   DATA[823,17] := 1.0;
   DATA[823,18] := 1.0;
   DATA[823,19] := 1.0;
   DATA[823,20] := 148.808;
   DATA[823,21] := 155.5755;
   DATA[823,22] := 1.717489;
   DATA[823,23] := 970.0205;
   DATA[823,24] := 2.0;
   DATA[823,25] := 2.0;
   DATA[823,26] := 7.878942;
   DATA[823,27] := 144.7578;
   DATA[823,28] := 263.0415;
   DATA[823,29] := 12.11228;
   DATA[823,30] := 1.72507;
   DATA[823,31] := 1.291918;
   DATA[823,32] := 0.7352687;
   DATA[823,33] := 0.3083624;
   DATA[823,34] := 2.0;
   DATA[823,35] := 250.5608;
   DATA[823,36] := 1.730048;
   DATA[823,37] := 189.4386;
   DATA[823,38] := 0.000128152;
   DATA[823,39] := 1.0;
   DATA[824,0] := 2.535311;
   DATA[824,1] := 568.1444;
   DATA[824,2] := 2.0;
   DATA[824,3] := 1.0;
   DATA[824,4] := 262.3366;
   DATA[824,5] := 8.46533;
   DATA[824,6] := 315.1243;
   DATA[824,8] := 1.0;
   DATA[824,9] := 1.0;
   DATA[824,10] := 1.0;
   DATA[824,11] := 2.032781;
   DATA[824,13] := 1010.118;
   DATA[824,14] := 1.0;
   DATA[824,15] := 1.0;
   DATA[824,16] := 1.0;
   DATA[824,17] := 1.0;
   DATA[824,18] := 1.0;
   DATA[824,19] := 1.0;
   DATA[824,20] := 148.808;
   DATA[824,21] := 155.5755;
   DATA[824,22] := 1.717489;
   DATA[824,23] := 970.0974;
   DATA[824,24] := 2.0;
   DATA[824,25] := 2.0;
   DATA[824,26] := 7.878942;
   DATA[824,27] := 144.7578;
   DATA[824,28] := 263.0415;
   DATA[824,29] := 12.11228;
   DATA[824,30] := 1.72507;
   DATA[824,31] := 1.291533;
   DATA[824,32] := 0.7352687;
   DATA[824,33] := 0.3083624;
   DATA[824,34] := 2.0;
   DATA[824,35] := 250.5768;
   DATA[824,36] := 1.730048;
   DATA[824,37] := 189.4386;
   DATA[824,38] := 0.000128152;
   DATA[824,39] := 1.0;
   DATA[825,0] := 2.535311;
   DATA[825,1] := 569.5575;
   DATA[825,2] := 2.0;
   DATA[825,3] := 1.0;
   DATA[825,4] := 262.3366;
   DATA[825,5] := 8.46533;
   DATA[825,6] := 315.1243;
   DATA[825,8] := 1.0;
   DATA[825,9] := 1.0;
   DATA[825,10] := 1.0;
   DATA[825,11] := 2.032781;
   DATA[825,13] := 1010.158;
   DATA[825,14] := 1.0;
   DATA[825,15] := 1.0;
   DATA[825,16] := 1.0;
   DATA[825,17] := 1.0;
   DATA[825,18] := 1.0;
   DATA[825,19] := 1.0;
   DATA[825,20] := 148.808;
   DATA[825,21] := 155.5755;
   DATA[825,22] := 1.717489;
   DATA[825,23] := 969.3668;
   DATA[825,24] := 2.0;
   DATA[825,25] := 2.0;
   DATA[825,26] := 7.878942;
   DATA[825,27] := 144.7578;
   DATA[825,28] := 263.0415;
   DATA[825,29] := 11.92002;
   DATA[825,30] := 1.72507;
   DATA[825,31] := 1.274881;
   DATA[825,32] := 0.7352687;
   DATA[825,33] := 0.3071454;
   DATA[825,34] := 2.0;
   DATA[825,35] := 250.721;
   DATA[825,36] := 1.730048;
   DATA[825,37] := 189.4386;
   DATA[825,38] := 0.000128152;
   DATA[825,39] := 1.0;
   DATA[826,0] := 2.544278;
   DATA[826,1] := 570.3426;
   DATA[826,2] := 2.0;
   DATA[826,3] := 1.0;
   DATA[826,4] := 262.3366;
   DATA[826,5] := 8.46533;
   DATA[826,6] := 315.1243;
   DATA[826,8] := 1.0;
   DATA[826,9] := 1.0;
   DATA[826,10] := 1.0;
   DATA[826,11] := 2.032781;
   DATA[826,13] := 1010.478;
   DATA[826,14] := 1.0;
   DATA[826,15] := 1.0;
   DATA[826,16] := 1.0;
   DATA[826,17] := 1.0;
   DATA[826,18] := 1.0;
   DATA[826,19] := 1.0;
   DATA[826,20] := 148.808;
   DATA[826,21] := 155.5755;
   DATA[826,22] := 1.717489;
   DATA[826,23] := 969.2515;
   DATA[826,24] := 2.0;
   DATA[826,25] := 2.0;
   DATA[826,26] := 7.878942;
   DATA[826,27] := 144.7578;
   DATA[826,28] := 263.0415;
   DATA[826,29] := 11.92002;
   DATA[826,30] := 1.72789;
   DATA[826,31] := 1.27898;
   DATA[826,32] := 0.7352687;
   DATA[826,33] := 0.3069532;
   DATA[826,34] := 2.0;
   DATA[826,35] := 250.721;
   DATA[826,36] := 1.730048;
   DATA[826,37] := 189.4386;
   DATA[826,38] := 0.000128152;
   DATA[826,39] := 1.0;
   DATA[827,0] := 2.547161;
   DATA[827,1] := 570.9706;
   DATA[827,2] := 2.0;
   DATA[827,3] := 1.0;
   DATA[827,4] := 262.3366;
   DATA[827,5] := 8.46533;
   DATA[827,6] := 315.1243;
   DATA[827,8] := 1.0;
   DATA[827,9] := 1.0;
   DATA[827,10] := 1.0;
   DATA[827,11] := 2.032781;
   DATA[827,13] := 1010.358;
   DATA[827,14] := 1.0;
   DATA[827,15] := 1.0;
   DATA[827,16] := 1.0;
   DATA[827,17] := 1.0;
   DATA[827,18] := 1.0;
   DATA[827,19] := 1.0;
   DATA[827,20] := 148.808;
   DATA[827,21] := 155.5755;
   DATA[827,22] := 1.719156;
   DATA[827,23] := 969.0208;
   DATA[827,24] := 2.0;
   DATA[827,25] := 2.0;
   DATA[827,26] := 7.878942;
   DATA[827,27] := 144.7578;
   DATA[827,28] := 263.0415;
   DATA[827,29] := 11.92002;
   DATA[827,30] := 1.728147;
   DATA[827,31] := 1.282183;
   DATA[827,32] := 0.7352687;
   DATA[827,33] := 0.3069532;
   DATA[827,34] := 2.0;
   DATA[827,35] := 250.721;
   DATA[827,36] := 1.730048;
   DATA[827,37] := 189.4386;
   DATA[827,38] := 0.000128152;
   DATA[827,39] := 1.0;
   DATA[828,0] := 2.547161;
   DATA[828,1] := 572.2659;
   DATA[828,2] := 2.0;
   DATA[828,3] := 1.0;
   DATA[828,4] := 262.3366;
   DATA[828,5] := 8.46533;
   DATA[828,6] := 315.1243;
   DATA[828,8] := 1.0;
   DATA[828,9] := 1.0;
   DATA[828,10] := 1.0;
   DATA[828,11] := 2.032781;
   DATA[828,13] := 1010.879;
   DATA[828,14] := 1.0;
   DATA[828,15] := 1.0;
   DATA[828,16] := 1.0;
   DATA[828,17] := 1.0;
   DATA[828,18] := 1.0;
   DATA[828,19] := 1.0;
   DATA[828,20] := 148.808;
   DATA[828,21] := 155.5755;
   DATA[828,22] := 1.719156;
   DATA[828,23] := 968.3671;
   DATA[828,24] := 2.0;
   DATA[828,25] := 2.0;
   DATA[828,26] := 7.878942;
   DATA[828,27] := 144.7578;
   DATA[828,28] := 263.0415;
   DATA[828,29] := 11.92002;
   DATA[828,30] := 1.728147;
   DATA[828,31] := 1.282183;
   DATA[828,32] := 0.7352687;
   DATA[828,33] := 0.3069532;
   DATA[828,34] := 2.0;
   DATA[828,35] := 250.721;
   DATA[828,36] := 1.730048;
   DATA[828,37] := 189.4386;
   DATA[828,38] := 0.000128152;
   DATA[828,39] := 1.0;
   DATA[829,0] := 2.547161;
   DATA[829,1] := 572.7762;
   DATA[829,2] := 2.0;
   DATA[829,3] := 1.0;
   DATA[829,4] := 262.3366;
   DATA[829,5] := 8.46533;
   DATA[829,6] := 315.1243;
   DATA[829,8] := 1.0;
   DATA[829,9] := 1.0;
   DATA[829,10] := 1.0;
   DATA[829,11] := 2.032781;
   DATA[829,13] := 1010.558;
   DATA[829,14] := 1.0;
   DATA[829,15] := 1.0;
   DATA[829,16] := 1.0;
   DATA[829,17] := 1.0;
   DATA[829,18] := 1.0;
   DATA[829,19] := 1.0;
   DATA[829,20] := 148.808;
   DATA[829,21] := 155.8062;
   DATA[829,22] := 1.719156;
   DATA[829,23] := 967.9056;
   DATA[829,24] := 2.0;
   DATA[829,25] := 2.0;
   DATA[829,26] := 7.878942;
   DATA[829,27] := 144.7578;
   DATA[829,28] := 263.0415;
   DATA[829,29] := 11.92002;
   DATA[829,30] := 1.729557;
   DATA[829,31] := 1.282183;
   DATA[829,32] := 0.7352687;
   DATA[829,33] := 0.3065689;
   DATA[829,34] := 2.0;
   DATA[829,35] := 250.721;
   DATA[829,36] := 1.730048;
   DATA[829,37] := 189.4386;
   DATA[829,38] := 0.000128152;
   DATA[829,39] := 1.0;
   DATA[830,0] := 2.547161;
   DATA[830,1] := 573.2473;
   DATA[830,2] := 2.0;
   DATA[830,3] := 1.0;
   DATA[830,4] := 262.3366;
   DATA[830,5] := 8.46533;
   DATA[830,6] := 315.1243;
   DATA[830,8] := 1.0;
   DATA[830,9] := 1.0;
   DATA[830,10] := 1.0;
   DATA[830,11] := 2.032781;
   DATA[830,13] := 1010.919;
   DATA[830,14] := 1.0;
   DATA[830,15] := 1.0;
   DATA[830,16] := 1.0;
   DATA[830,17] := 1.0;
   DATA[830,18] := 1.0;
   DATA[830,19] := 1.0;
   DATA[830,20] := 148.808;
   DATA[830,21] := 155.8062;
   DATA[830,22] := 1.717746;
   DATA[830,23] := 967.4827;
   DATA[830,24] := 2.0;
   DATA[830,25] := 2.0;
   DATA[830,26] := 7.878942;
   DATA[830,27] := 144.7578;
   DATA[830,28] := 263.0415;
   DATA[830,29] := 11.92002;
   DATA[830,30] := 1.729557;
   DATA[830,31] := 1.282183;
   DATA[830,32] := 0.7352687;
   DATA[830,33] := 0.3079781;
   DATA[830,34] := 2.0;
   DATA[830,35] := 250.4967;
   DATA[830,36] := 1.730048;
   DATA[830,37] := 189.4386;
   DATA[830,38] := 0.000128152;
   DATA[830,39] := 1.0;
   DATA[831,0] := 2.547161;
   DATA[831,1] := 573.3258;
   DATA[831,2] := 2.0;
   DATA[831,3] := 1.0;
   DATA[831,4] := 262.3366;
   DATA[831,5] := 8.46533;
   DATA[831,6] := 315.1243;
   DATA[831,8] := 1.0;
   DATA[831,9] := 1.0;
   DATA[831,10] := 1.0;
   DATA[831,11] := 2.032781;
   DATA[831,13] := 1010.718;
   DATA[831,14] := 1.0;
   DATA[831,15] := 1.0;
   DATA[831,16] := 1.0;
   DATA[831,17] := 1.0;
   DATA[831,18] := 1.0;
   DATA[831,19] := 1.0;
   DATA[831,20] := 148.808;
   DATA[831,21] := 155.8062;
   DATA[831,22] := 1.717746;
   DATA[831,23] := 967.3289;
   DATA[831,24] := 2.0;
   DATA[831,25] := 2.0;
   DATA[831,26] := 7.878942;
   DATA[831,27] := 144.7578;
   DATA[831,28] := 263.0415;
   DATA[831,29] := 11.92002;
   DATA[831,30] := 1.729557;
   DATA[831,31] := 1.271935;
   DATA[831,32] := 0.7352687;
   DATA[831,33] := 0.3083624;
   DATA[831,34] := 2.0;
   DATA[831,35] := 250.4967;
   DATA[831,36] := 1.730048;
   DATA[831,37] := 189.4386;
   DATA[831,38] := 0.000128152;
   DATA[831,39] := 1.0;
   DATA[832,0] := 2.547161;
   DATA[832,1] := 574.4249;
   DATA[832,2] := 2.0;
   DATA[832,3] := 1.0;
   DATA[832,4] := 262.3366;
   DATA[832,5] := 8.46533;
   DATA[832,6] := 315.1243;
   DATA[832,8] := 1.0;
   DATA[832,9] := 1.0;
   DATA[832,10] := 1.0;
   DATA[832,11] := 2.032781;
   DATA[832,13] := 1011.039;
   DATA[832,14] := 1.0;
   DATA[832,15] := 1.0;
   DATA[832,16] := 1.0;
   DATA[832,17] := 1.0;
   DATA[832,18] := 1.0;
   DATA[832,19] := 1.0;
   DATA[832,20] := 148.808;
   DATA[832,21] := 155.5755;
   DATA[832,22] := 1.717746;
   DATA[832,23] := 966.9059;
   DATA[832,24] := 2.0;
   DATA[832,25] := 2.0;
   DATA[832,26] := 7.878942;
   DATA[832,27] := 144.7578;
   DATA[832,28] := 263.0415;
   DATA[832,29] := 11.92002;
   DATA[832,30] := 1.729557;
   DATA[832,31] := 1.279621;
   DATA[832,32] := 0.7352687;
   DATA[832,33] := 0.3083624;
   DATA[832,34] := 2.0;
   DATA[832,35] := 250.4967;
   DATA[832,36] := 1.730048;
   DATA[832,37] := 189.4386;
   DATA[832,38] := 0.000128152;
   DATA[832,39] := 1.0;
   DATA[833,0] := 2.555168;
   DATA[833,1] := 575.4454;
   DATA[833,2] := 2.0;
   DATA[833,3] := 1.0;
   DATA[833,4] := 262.3366;
   DATA[833,5] := 8.46533;
   DATA[833,6] := 315.1243;
   DATA[833,8] := 1.0;
   DATA[833,9] := 1.0;
   DATA[833,10] := 1.0;
   DATA[833,11] := 2.032781;
   DATA[833,13] := 1010.959;
   DATA[833,14] := 1.0;
   DATA[833,15] := 1.0;
   DATA[833,16] := 1.0;
   DATA[833,17] := 1.0;
   DATA[833,18] := 1.0;
   DATA[833,19] := 1.0;
   DATA[833,20] := 148.808;
   DATA[833,21] := 155.5755;
   DATA[833,22] := 1.717746;
   DATA[833,23] := 966.6752;
   DATA[833,24] := 2.0;
   DATA[833,25] := 2.0;
   DATA[833,26] := 7.878942;
   DATA[833,27] := 144.7578;
   DATA[833,28] := 263.0415;
   DATA[833,29] := 12.15073;
   DATA[833,30] := 1.729557;
   DATA[833,31] := 1.290893;
   DATA[833,32] := 0.7352687;
   DATA[833,33] := 0.3083624;
   DATA[833,34] := 2.0;
   DATA[833,35] := 250.737;
   DATA[833,36] := 1.730048;
   DATA[833,37] := 189.4386;
   DATA[833,38] := 0.000128152;
   DATA[833,39] := 1.0;
   DATA[834,0] := 2.555168;
   DATA[834,1] := 576.2697;
   DATA[834,2] := 2.0;
   DATA[834,3] := 1.0;
   DATA[834,4] := 262.3366;
   DATA[834,5] := 8.46533;
   DATA[834,6] := 315.1243;
   DATA[834,8] := 1.0;
   DATA[834,9] := 1.0;
   DATA[834,10] := 1.0;
   DATA[834,11] := 2.032781;
   DATA[834,13] := 1011.279;
   DATA[834,14] := 1.0;
   DATA[834,15] := 1.0;
   DATA[834,16] := 1.0;
   DATA[834,17] := 1.0;
   DATA[834,18] := 1.0;
   DATA[834,19] := 1.0;
   DATA[834,20] := 148.808;
   DATA[834,21] := 155.5755;
   DATA[834,22] := 1.717746;
   DATA[834,23] := 966.3676;
   DATA[834,24] := 2.0;
   DATA[834,25] := 2.0;
   DATA[834,26] := 7.878942;
   DATA[834,27] := 144.7578;
   DATA[834,28] := 263.0415;
   DATA[834,29] := 12.15073;
   DATA[834,30] := 1.729557;
   DATA[834,31] := 1.286153;
   DATA[834,32] := 0.7352687;
   DATA[834,33] := 0.3083624;
   DATA[834,34] := 2.0;
   DATA[834,35] := 250.737;
   DATA[834,36] := 1.730048;
   DATA[834,37] := 189.4386;
   DATA[834,38] := 0.000128152;
   DATA[834,39] := 1.0;
   DATA[835,0] := 2.555168;
   DATA[835,1] := 577.251;
   DATA[835,2] := 2.0;
   DATA[835,3] := 1.0;
   DATA[835,4] := 262.3366;
   DATA[835,5] := 8.46533;
   DATA[835,6] := 315.1243;
   DATA[835,8] := 1.0;
   DATA[835,9] := 1.0;
   DATA[835,10] := 1.0;
   DATA[835,11] := 2.032781;
   DATA[835,13] := 1011.079;
   DATA[835,14] := 1.0;
   DATA[835,15] := 1.0;
   DATA[835,16] := 1.0;
   DATA[835,17] := 1.0;
   DATA[835,18] := 1.0;
   DATA[835,19] := 1.0;
   DATA[835,20] := 148.808;
   DATA[835,21] := 155.5755;
   DATA[835,22] := 1.717746;
   DATA[835,23] := 965.7139;
   DATA[835,24] := 2.0;
   DATA[835,25] := 2.0;
   DATA[835,26] := 7.878942;
   DATA[835,27] := 144.7578;
   DATA[835,28] := 263.0415;
   DATA[835,29] := 12.15073;
   DATA[835,30] := 1.7293;
   DATA[835,31] := 1.288715;
   DATA[835,32] := 0.7352687;
   DATA[835,33] := 0.3083624;
   DATA[835,34] := 2.0;
   DATA[835,35] := 250.737;
   DATA[835,36] := 1.730048;
   DATA[835,37] := 189.6949;
   DATA[835,38] := 0.000128152;
   DATA[835,39] := 1.0;
   DATA[836,0] := 2.555168;
   DATA[836,1] := 577.8006;
   DATA[836,2] := 2.0;
   DATA[836,3] := 1.0;
   DATA[836,4] := 262.3366;
   DATA[836,5] := 8.46533;
   DATA[836,6] := 315.1243;
   DATA[836,8] := 1.0;
   DATA[836,9] := 1.0;
   DATA[836,10] := 1.0;
   DATA[836,11] := 2.032781;
   DATA[836,13] := 1011.079;
   DATA[836,14] := 1.0;
   DATA[836,15] := 1.0;
   DATA[836,16] := 1.0;
   DATA[836,17] := 1.0;
   DATA[836,18] := 1.0;
   DATA[836,19] := 1.0;
   DATA[836,20] := 148.808;
   DATA[836,21] := 155.5755;
   DATA[836,22] := 1.718515;
   DATA[836,23] := 965.3294;
   DATA[836,24] := 2.0;
   DATA[836,25] := 2.0;
   DATA[836,26] := 7.878942;
   DATA[836,27] := 144.7578;
   DATA[836,28] := 263.0415;
   DATA[836,29] := 12.15073;
   DATA[836,30] := 1.7293;
   DATA[836,31] := 1.281542;
   DATA[836,32] := 0.7352687;
   DATA[836,33] := 0.3083624;
   DATA[836,34] := 2.0;
   DATA[836,35] := 250.8972;
   DATA[836,36] := 1.730048;
   DATA[836,37] := 189.6949;
   DATA[836,38] := 0.000128152;
   DATA[836,39] := 1.0;
   DATA[837,0] := 2.555168;
   DATA[837,1] := 578.8212;
   DATA[837,2] := 2.0;
   DATA[837,3] := 1.0;
   DATA[837,4] := 262.3366;
   DATA[837,5] := 8.46533;
   DATA[837,6] := 315.1243;
   DATA[837,8] := 1.0;
   DATA[837,9] := 1.0;
   DATA[837,10] := 1.0;
   DATA[837,11] := 2.032781;
   DATA[837,13] := 1011.239;
   DATA[837,14] := 1.0;
   DATA[837,15] := 1.0;
   DATA[837,16] := 1.0;
   DATA[837,17] := 1.0;
   DATA[837,18] := 1.0;
   DATA[837,19] := 1.0;
   DATA[837,20] := 148.808;
   DATA[837,21] := 155.5755;
   DATA[837,22] := 1.720565;
   DATA[837,23] := 964.6373;
   DATA[837,24] := 2.0;
   DATA[837,25] := 2.0;
   DATA[837,26] := 7.878942;
   DATA[837,27] := 144.7578;
   DATA[837,28] := 263.0415;
   DATA[837,29] := 12.15073;
   DATA[837,30] := 1.7293;
   DATA[837,31] := 1.272192;
   DATA[837,32] := 0.7352687;
   DATA[837,33] := 0.3083624;
   DATA[837,34] := 2.0;
   DATA[837,35] := 250.8972;
   DATA[837,36] := 1.730048;
   DATA[837,37] := 189.6949;
   DATA[837,38] := 0.000128152;
   DATA[837,39] := 1.0;
   DATA[838,0] := 2.553886;
   DATA[838,1] := 579.724;
   DATA[838,2] := 2.0;
   DATA[838,3] := 1.0;
   DATA[838,4] := 262.3366;
   DATA[838,5] := 8.46533;
   DATA[838,6] := 315.1243;
   DATA[838,8] := 1.0;
   DATA[838,9] := 1.0;
   DATA[838,10] := 1.0;
   DATA[838,11] := 2.032781;
   DATA[838,13] := 1011.279;
   DATA[838,14] := 1.0;
   DATA[838,15] := 1.0;
   DATA[838,16] := 1.0;
   DATA[838,17] := 1.0;
   DATA[838,18] := 1.0;
   DATA[838,19] := 1.0;
   DATA[838,20] := 148.808;
   DATA[838,21] := 155.5755;
   DATA[838,22] := 1.720565;
   DATA[838,23] := 964.5988;
   DATA[838,24] := 2.0;
   DATA[838,25] := 2.0;
   DATA[838,26] := 7.878942;
   DATA[838,27] := 144.7578;
   DATA[838,28] := 263.0415;
   DATA[838,29] := 12.15073;
   DATA[838,30] := 1.7293;
   DATA[838,31] := 1.271679;
   DATA[838,32] := 0.736421;
   DATA[838,33] := 0.3083624;
   DATA[838,34] := 2.0;
   DATA[838,35] := 250.8972;
   DATA[838,36] := 1.730048;
   DATA[838,37] := 189.6949;
   DATA[838,38] := 0.000128152;
   DATA[838,39] := 1.0;
   DATA[839,0] := 2.54684;
   DATA[839,1] := 580.7053;
   DATA[839,2] := 2.0;
   DATA[839,3] := 1.0;
   DATA[839,4] := 262.3366;
   DATA[839,5] := 8.46533;
   DATA[839,6] := 315.1243;
   DATA[839,8] := 1.0;
   DATA[839,9] := 1.0;
   DATA[839,10] := 1.0;
   DATA[839,11] := 2.032781;
   DATA[839,13] := 1011.079;
   DATA[839,14] := 1.0;
   DATA[839,15] := 1.0;
   DATA[839,16] := 1.0;
   DATA[839,17] := 1.0;
   DATA[839,18] := 1.0;
   DATA[839,19] := 1.0;
   DATA[839,20] := 148.808;
   DATA[839,21] := 155.5755;
   DATA[839,22] := 1.720565;
   DATA[839,23] := 964.1758;
   DATA[839,24] := 2.0;
   DATA[839,25] := 2.0;
   DATA[839,26] := 7.878942;
   DATA[839,27] := 144.7578;
   DATA[839,28] := 263.0415;
   DATA[839,29] := 12.15073;
   DATA[839,30] := 1.7293;
   DATA[839,31] := 1.271551;
   DATA[839,32] := 0.7366771;
   DATA[839,33] := 0.3068891;
   DATA[839,34] := 2.0;
   DATA[839,35] := 250.8972;
   DATA[839,36] := 1.730048;
   DATA[839,37] := 189.5668;
   DATA[839,38] := 0.000128152;
   DATA[839,39] := 1.0;
   DATA[840,0] := 2.542356;
   DATA[840,1] := 581.2941;
   DATA[840,2] := 2.0;
   DATA[840,3] := 1.0;
   DATA[840,4] := 262.3366;
   DATA[840,5] := 8.46533;
   DATA[840,6] := 315.1243;
   DATA[840,8] := 1.0;
   DATA[840,9] := 1.0;
   DATA[840,10] := 1.0;
   DATA[840,11] := 2.026378;
   DATA[840,13] := 1010.879;
   DATA[840,14] := 1.0;
   DATA[840,15] := 1.0;
   DATA[840,16] := 1.0;
   DATA[840,17] := 1.0;
   DATA[840,18] := 1.0;
   DATA[840,19] := 1.0;
   DATA[840,20] := 148.808;
   DATA[840,21] := 155.5755;
   DATA[840,22] := 1.718771;
   DATA[840,23] := 963.7529;
   DATA[840,24] := 2.0;
   DATA[840,25] := 2.0;
   DATA[840,26] := 7.878942;
   DATA[840,27] := 144.7578;
   DATA[840,28] := 263.0415;
   DATA[840,29] := 12.15073;
   DATA[840,30] := 1.728019;
   DATA[840,31] := 1.271551;
   DATA[840,32] := 0.7373172;
   DATA[840,33] := 0.3068891;
   DATA[840,34] := 2.0;
   DATA[840,35] := 250.785;
   DATA[840,36] := 1.730048;
   DATA[840,37] := 189.4546;
   DATA[840,38] := 0.000128152;
   DATA[840,39] := 1.0;
   DATA[841,0] := 2.538833;
   DATA[841,1] := 581.5688;
   DATA[841,2] := 2.0;
   DATA[841,3] := 1.0;
   DATA[841,4] := 262.3366;
   DATA[841,5] := 8.46501;
   DATA[841,6] := 315.1243;
   DATA[841,8] := 1.0;
   DATA[841,9] := 1.0;
   DATA[841,10] := 1.0;
   DATA[841,11] := 2.026378;
   DATA[841,13] := 1011.159;
   DATA[841,14] := 1.0;
   DATA[841,15] := 1.0;
   DATA[841,16] := 1.0;
   DATA[841,17] := 1.0;
   DATA[841,18] := 1.0;
   DATA[841,19] := 1.0;
   DATA[841,20] := 148.808;
   DATA[841,21] := 155.5755;
   DATA[841,22] := 1.718771;
   DATA[841,23] := 963.4068;
   DATA[841,24] := 2.0;
   DATA[841,25] := 2.0;
   DATA[841,26] := 7.878942;
   DATA[841,27] := 144.7578;
   DATA[841,28] := 263.0415;
   DATA[841,29] := 12.15073;
   DATA[841,30] := 1.726609;
   DATA[841,31] := 1.271551;
   DATA[841,32] := 0.7383414;
   DATA[841,33] := 0.3068891;
   DATA[841,34] := 2.0;
   DATA[841,35] := 250.4807;
   DATA[841,36] := 1.730048;
   DATA[841,37] := 189.1983;
   DATA[841,38] := 0.000128152;
   DATA[841,39] := 1.0;
   DATA[842,0] := 2.538833;
   DATA[842,1] := 581.5688;
   DATA[842,2] := 2.0;
   DATA[842,3] := 1.0;
   DATA[842,4] := 262.3366;
   DATA[842,5] := 8.46501;
   DATA[842,6] := 315.1243;
   DATA[842,8] := 1.0;
   DATA[842,9] := 1.0;
   DATA[842,10] := 1.0;
   DATA[842,11] := 2.026378;
   DATA[842,13] := 1011.159;
   DATA[842,14] := 1.0;
   DATA[842,15] := 1.0;
   DATA[842,16] := 1.0;
   DATA[842,17] := 1.0;
   DATA[842,18] := 1.0;
   DATA[842,19] := 1.0;
   DATA[842,20] := 148.808;
   DATA[842,21] := 155.5755;
   DATA[842,22] := 1.718771;
   DATA[842,23] := 963.4068;
   DATA[842,24] := 2.0;
   DATA[842,25] := 2.0;
   DATA[842,26] := 7.878942;
   DATA[842,27] := 144.7578;
   DATA[842,28] := 263.0415;
   DATA[842,29] := 12.15073;
   DATA[842,30] := 1.726609;
   DATA[842,31] := 1.271551;
   DATA[842,32] := 0.7383414;
   DATA[842,33] := 0.3068891;
   DATA[842,34] := 2.0;
   DATA[842,35] := 250.4807;
   DATA[842,36] := 1.730048;
   DATA[842,37] := 189.1983;
   DATA[842,38] := 0.000128152;
   DATA[842,39] := 1.0;
   DATA[843,0] := 2.536912;
   DATA[843,1] := 581.9614;
   DATA[843,2] := 2.0;
   DATA[843,3] := 1.0;
   DATA[843,4] := 262.3366;
   DATA[843,5] := 8.462446;
   DATA[843,6] := 315.1243;
   DATA[843,8] := 1.0;
   DATA[843,9] := 1.0;
   DATA[843,10] := 1.0;
   DATA[843,11] := 2.026378;
   DATA[843,13] := 1011.039;
   DATA[843,14] := 1.0;
   DATA[843,15] := 1.0;
   DATA[843,16] := 1.0;
   DATA[843,17] := 1.0;
   DATA[843,18] := 1.0;
   DATA[843,19] := 1.0;
   DATA[843,20] := 148.808;
   DATA[843,21] := 155.5499;
   DATA[843,22] := 1.718771;
   DATA[843,23] := 963.2914;
   DATA[843,24] := 2.0;
   DATA[843,25] := 2.0;
   DATA[843,26] := 7.878942;
   DATA[843,27] := 144.7578;
   DATA[843,28] := 263.0415;
   DATA[843,29] := 12.15073;
   DATA[843,30] := 1.726609;
   DATA[843,31] := 1.281158;
   DATA[843,32] := 0.7368051;
   DATA[843,33] := 0.3068891;
   DATA[843,34] := 2.0;
   DATA[843,35] := 250.4807;
   DATA[843,36] := 1.730048;
   DATA[843,37] := 189.1983;
   DATA[843,38] := 0.000128152;
   DATA[843,39] := 1.0;
   DATA[844,0] := 2.544278;
   DATA[844,1] := 582.1577;
   DATA[844,2] := 2.0;
   DATA[844,3] := 1.0;
   DATA[844,4] := 262.3366;
   DATA[844,5] := 8.462446;
   DATA[844,6] := 315.1243;
   DATA[844,8] := 1.0;
   DATA[844,9] := 1.0;
   DATA[844,10] := 1.0;
   DATA[844,11] := 2.026378;
   DATA[844,13] := 1011.359;
   DATA[844,14] := 1.0;
   DATA[844,15] := 1.0;
   DATA[844,16] := 1.0;
   DATA[844,17] := 1.0;
   DATA[844,18] := 1.0;
   DATA[844,19] := 1.0;
   DATA[844,20] := 148.808;
   DATA[844,21] := 155.5242;
   DATA[844,22] := 1.718771;
   DATA[844,23] := 962.8685;
   DATA[844,24] := 2.0;
   DATA[844,25] := 2.0;
   DATA[844,26] := 7.878942;
   DATA[844,27] := 144.7578;
   DATA[844,28] := 263.0415;
   DATA[844,29] := 12.15073;
   DATA[844,30] := 1.725968;
   DATA[844,31] := 1.281927;
   DATA[844,32] := 0.7352687;
   DATA[844,33] := 0.3068891;
   DATA[844,34] := 2.0;
   DATA[844,35] := 250.4807;
   DATA[844,36] := 1.730048;
   DATA[844,37] := 189.1983;
   DATA[844,38] := 0.000128152;
   DATA[844,39] := 1.0;
   DATA[845,0] := 2.54588;
   DATA[845,1] := 582.5109;
   DATA[845,2] := 2.0;
   DATA[845,3] := 1.0;
   DATA[845,4] := 262.3366;
   DATA[845,5] := 8.462446;
   DATA[845,6] := 315.1243;
   DATA[845,8] := 1.0;
   DATA[845,9] := 1.0;
   DATA[845,10] := 1.0;
   DATA[845,11] := 2.026378;
   DATA[845,13] := 1011.119;
   DATA[845,14] := 1.0;
   DATA[845,15] := 1.0;
   DATA[845,16] := 1.0;
   DATA[845,17] := 1.0;
   DATA[845,18] := 1.0;
   DATA[845,19] := 1.0;
   DATA[845,20] := 148.808;
   DATA[845,21] := 155.3448;
   DATA[845,22] := 1.71467;
   DATA[845,23] := 962.1379;
   DATA[845,24] := 2.0;
   DATA[845,25] := 2.0;
   DATA[845,26] := 7.878942;
   DATA[845,27] := 144.7578;
   DATA[845,28] := 263.0415;
   DATA[845,29] := 12.07383;
   DATA[845,30] := 1.725327;
   DATA[845,31] := 1.282439;
   DATA[845,32] := 0.7352687;
   DATA[845,33] := 0.3084265;
   DATA[845,34] := 2.0;
   DATA[845,35] := 250.3845;
   DATA[845,36] := 1.730048;
   DATA[845,37] := 189.1983;
   DATA[845,38] := 0.000128152;
   DATA[845,39] := 1.0;
   DATA[846,0] := 2.54588;
   DATA[846,1] := 582.7465;
   DATA[846,2] := 2.0;
   DATA[846,3] := 1.0;
   DATA[846,4] := 262.3366;
   DATA[846,5] := 8.462446;
   DATA[846,6] := 315.1243;
   DATA[846,8] := 1.0;
   DATA[846,9] := 1.0;
   DATA[846,10] := 1.0;
   DATA[846,11] := 2.026378;
   DATA[846,13] := 1011.159;
   DATA[846,14] := 1.0;
   DATA[846,15] := 1.0;
   DATA[846,16] := 1.0;
   DATA[846,17] := 1.0;
   DATA[846,18] := 1.0;
   DATA[846,19] := 1.0;
   DATA[846,20] := 148.808;
   DATA[846,21] := 155.3448;
   DATA[846,22] := 1.713901;
   DATA[846,23] := 961.6381;
   DATA[846,24] := 2.0;
   DATA[846,25] := 2.0;
   DATA[846,26] := 7.878942;
   DATA[846,27] := 144.7578;
   DATA[846,28] := 263.0415;
   DATA[846,29] := 12.07383;
   DATA[846,30] := 1.725327;
   DATA[846,31] := 1.282439;
   DATA[846,32] := 0.7352687;
   DATA[846,33] := 0.3084265;
   DATA[846,34] := 2.0;
   DATA[846,35] := 250.2243;
   DATA[846,36] := 1.730048;
   DATA[846,37] := 188.958;
   DATA[846,38] := 0.000128152;
   DATA[846,39] := 1.0;
   DATA[847,0] := 2.54588;
   DATA[847,1] := 582.9034;
   DATA[847,2] := 2.0;
   DATA[847,3] := 1.0;
   DATA[847,4] := 262.3366;
   DATA[847,5] := 8.462446;
   DATA[847,6] := 315.1243;
   DATA[847,8] := 1.0;
   DATA[847,9] := 1.0;
   DATA[847,10] := 1.0;
   DATA[847,11] := 2.026378;
   DATA[847,13] := 1010.959;
   DATA[847,14] := 1.0;
   DATA[847,15] := 1.0;
   DATA[847,16] := 1.0;
   DATA[847,17] := 1.0;
   DATA[847,18] := 1.0;
   DATA[847,19] := 1.0;
   DATA[847,20] := 148.808;
   DATA[847,21] := 155.3448;
   DATA[847,22] := 1.713901;
   DATA[847,23] := 960.9844;
   DATA[847,24] := 2.0;
   DATA[847,25] := 2.0;
   DATA[847,26] := 7.878942;
   DATA[847,27] := 144.7578;
   DATA[847,28] := 263.0415;
   DATA[847,29] := 12.07383;
   DATA[847,30] := 1.725327;
   DATA[847,31] := 1.268349;
   DATA[847,32] := 0.7352687;
   DATA[847,33] := 0.3084265;
   DATA[847,34] := 2.0;
   DATA[847,35] := 250.2243;
   DATA[847,36] := 1.730048;
   DATA[847,37] := 188.958;
   DATA[847,38] := 0.000128152;
   DATA[847,39] := 1.0;
   DATA[848,0] := 2.551324;
   DATA[848,1] := 583.139;
   DATA[848,2] := 2.0;
   DATA[848,3] := 1.0;
   DATA[848,4] := 262.3366;
   DATA[848,5] := 8.462446;
   DATA[848,6] := 315.1243;
   DATA[848,8] := 1.0;
   DATA[848,9] := 1.0;
   DATA[848,10] := 1.0;
   DATA[848,11] := 2.026378;
   DATA[848,13] := 1010.718;
   DATA[848,14] := 1.0;
   DATA[848,15] := 1.0;
   DATA[848,16] := 1.0;
   DATA[848,17] := 1.0;
   DATA[848,18] := 1.0;
   DATA[848,19] := 1.0;
   DATA[848,20] := 148.808;
   DATA[848,21] := 155.3448;
   DATA[848,22] := 1.713901;
   DATA[848,23] := 961.4458;
   DATA[848,24] := 2.0;
   DATA[848,25] := 2.0;
   DATA[848,26] := 7.878942;
   DATA[848,27] := 144.7578;
   DATA[848,28] := 263.0415;
   DATA[848,29] := 12.07383;
   DATA[848,30] := 1.724686;
   DATA[848,31] := 1.261432;
   DATA[848,32] := 0.7352687;
   DATA[848,33] := 0.3084265;
   DATA[848,34] := 2.0;
   DATA[848,35] := 250.2243;
   DATA[848,36] := 1.730048;
   DATA[848,37] := 188.958;
   DATA[848,38] := 0.000128152;
   DATA[848,39] := 1.0;
   DATA[849,0] := 2.551324;
   DATA[849,1] := 583.0997;
   DATA[849,2] := 2.0;
   DATA[849,3] := 1.0;
   DATA[849,4] := 262.3366;
   DATA[849,5] := 8.460844;
   DATA[849,6] := 315.1243;
   DATA[849,8] := 1.0;
   DATA[849,9] := 1.0;
   DATA[849,10] := 1.0;
   DATA[849,11] := 2.026378;
   DATA[849,13] := 1010.678;
   DATA[849,14] := 1.0;
   DATA[849,15] := 1.0;
   DATA[849,16] := 1.0;
   DATA[849,17] := 1.0;
   DATA[849,18] := 1.0;
   DATA[849,19] := 1.0;
   DATA[849,20] := 148.808;
   DATA[849,21] := 155.3448;
   DATA[849,22] := 1.713901;
   DATA[849,23] := 961.4843;
   DATA[849,24] := 2.0;
   DATA[849,25] := 2.0;
   DATA[849,26] := 7.878942;
   DATA[849,27] := 144.6039;
   DATA[849,28] := 263.0415;
   DATA[849,29] := 12.07383;
   DATA[849,30] := 1.724173;
   DATA[849,31] := 1.275138;
   DATA[849,32] := 0.7352687;
   DATA[849,33] := 0.3084265;
   DATA[849,34] := 2.0;
   DATA[849,35] := 250.2243;
   DATA[849,36] := 1.730048;
   DATA[849,37] := 189.022;
   DATA[849,38] := 0.000128152;
   DATA[849,39] := 1.0;
   DATA[850,0] := 2.551324;
   DATA[850,1] := 583.5707;
   DATA[850,2] := 2.0;
   DATA[850,3] := 1.0;
   DATA[850,4] := 262.3366;
   DATA[850,5] := 8.460203;
   DATA[850,6] := 315.1243;
   DATA[850,8] := 1.0;
   DATA[850,9] := 1.0;
   DATA[850,10] := 1.0;
   DATA[850,11] := 2.026378;
   DATA[850,13] := 1010.678;
   DATA[850,14] := 1.0;
   DATA[850,15] := 1.0;
   DATA[850,16] := 1.0;
   DATA[850,17] := 1.0;
   DATA[850,18] := 1.0;
   DATA[850,19] := 1.0;
   DATA[850,20] := 148.808;
   DATA[850,21] := 155.3448;
   DATA[850,22] := 1.713901;
   DATA[850,23] := 961.0613;
   DATA[850,24] := 2.0;
   DATA[850,25] := 2.0;
   DATA[850,26] := 7.878942;
   DATA[850,27] := 144.6039;
   DATA[850,28] := 263.0415;
   DATA[850,29] := 12.07383;
   DATA[850,30] := 1.724173;
   DATA[850,31] := 1.290765;
   DATA[850,32] := 0.7352687;
   DATA[850,33] := 0.3084265;
   DATA[850,34] := 2.0;
   DATA[850,35] := 250.5447;
   DATA[850,36] := 1.730048;
   DATA[850,37] := 189.2464;
   DATA[850,38] := 0.000128152;
   DATA[850,39] := 1.0;
   DATA[851,0] := 2.551324;
   DATA[851,1] := 584.5128;
   DATA[851,2] := 2.0;
   DATA[851,3] := 1.0;
   DATA[851,4] := 262.3366;
   DATA[851,5] := 8.460203;
   DATA[851,6] := 315.1243;
   DATA[851,8] := 1.0;
   DATA[851,9] := 1.0;
   DATA[851,10] := 1.0;
   DATA[851,11] := 2.026378;
   DATA[851,13] := 1010.879;
   DATA[851,14] := 1.0;
   DATA[851,15] := 1.0;
   DATA[851,16] := 1.0;
   DATA[851,17] := 1.0;
   DATA[851,18] := 1.0;
   DATA[851,19] := 1.0;
   DATA[851,20] := 148.808;
   DATA[851,21] := 155.3448;
   DATA[851,22] := 1.713901;
   DATA[851,23] := 960.6768;
   DATA[851,24] := 2.0;
   DATA[851,25] := 2.0;
   DATA[851,26] := 7.878942;
   DATA[851,27] := 144.6039;
   DATA[851,28] := 263.0415;
   DATA[851,29] := 12.07383;
   DATA[851,30] := 1.724173;
   DATA[851,31] := 1.291789;
   DATA[851,32] := 0.7352687;
   DATA[851,33] := 0.3084265;
   DATA[851,34] := 2.0;
   DATA[851,35] := 250.5447;
   DATA[851,36] := 1.730048;
   DATA[851,37] := 189.2784;
   DATA[851,38] := 0.000128152;
   DATA[851,39] := 1.0;
   DATA[852,0] := 2.547481;
   DATA[852,1] := 585.0624;
   DATA[852,2] := 2.0;
   DATA[852,3] := 1.0;
   DATA[852,4] := 262.3366;
   DATA[852,5] := 8.460203;
   DATA[852,6] := 315.1243;
   DATA[852,8] := 1.0;
   DATA[852,9] := 1.0;
   DATA[852,10] := 1.0;
   DATA[852,11] := 2.026378;
   DATA[852,13] := 1010.839;
   DATA[852,14] := 1.0;
   DATA[852,15] := 1.0;
   DATA[852,16] := 1.0;
   DATA[852,17] := 1.0;
   DATA[852,18] := 1.0;
   DATA[852,19] := 1.0;
   DATA[852,20] := 148.808;
   DATA[852,21] := 155.3448;
   DATA[852,22] := 1.715311;
   DATA[852,23] := 959.6385;
   DATA[852,24] := 2.0;
   DATA[852,25] := 2.0;
   DATA[852,26] := 7.878942;
   DATA[852,27] := 144.6039;
   DATA[852,28] := 263.0415;
   DATA[852,29] := 12.07383;
   DATA[852,30] := 1.725455;
   DATA[852,31] := 1.277187;
   DATA[852,32] := 0.7352687;
   DATA[852,33] := 0.3084265;
   DATA[852,34] := 2.0;
   DATA[852,35] := 250.5447;
   DATA[852,36] := 1.730048;
   DATA[852,37] := 189.4226;
   DATA[852,38] := 0.000128152;
   DATA[852,39] := 1.0;
   DATA[853,0] := 2.551645;
   DATA[853,1] := 585.2979;
   DATA[853,2] := 2.0;
   DATA[853,3] := 1.0;
   DATA[853,4] := 262.3366;
   DATA[853,5] := 8.460203;
   DATA[853,6] := 315.1243;
   DATA[853,8] := 1.0;
   DATA[853,9] := 1.0;
   DATA[853,10] := 1.0;
   DATA[853,11] := 2.026378;
   DATA[853,13] := 1011.159;
   DATA[853,14] := 1.0;
   DATA[853,15] := 1.0;
   DATA[853,16] := 1.0;
   DATA[853,17] := 1.0;
   DATA[853,18] := 1.0;
   DATA[853,19] := 1.0;
   DATA[853,20] := 148.808;
   DATA[853,21] := 155.3448;
   DATA[853,22] := 1.716592;
   DATA[853,23] := 959.2156;
   DATA[853,24] := 2.0;
   DATA[853,25] := 2.0;
   DATA[853,26] := 7.878942;
   DATA[853,27] := 144.6039;
   DATA[853,28] := 263.0415;
   DATA[853,29] := 12.07383;
   DATA[853,30] := 1.727506;
   DATA[853,31] := 1.261432;
   DATA[853,32] := 0.7352687;
   DATA[853,33] := 0.3079781;
   DATA[853,34] := 2.0;
   DATA[853,35] := 250.6729;
   DATA[853,36] := 1.730048;
   DATA[853,37] := 189.4226;
   DATA[853,38] := 0.000128152;
   DATA[853,39] := 1.0;
   DATA[854,0] := 2.555488;
   DATA[854,1] := 585.8082;
   DATA[854,2] := 2.0;
   DATA[854,3] := 1.0;
   DATA[854,4] := 262.3366;
   DATA[854,5] := 8.460203;
   DATA[854,6] := 315.1243;
   DATA[854,8] := 1.0;
   DATA[854,9] := 1.0;
   DATA[854,10] := 1.0;
   DATA[854,11] := 2.026378;
   DATA[854,13] := 1010.959;
   DATA[854,14] := 1.0;
   DATA[854,15] := 1.0;
   DATA[854,16] := 1.0;
   DATA[854,17] := 1.0;
   DATA[854,18] := 1.0;
   DATA[854,19] := 1.0;
   DATA[854,20] := 148.808;
   DATA[854,21] := 155.3448;
   DATA[854,22] := 1.716592;
   DATA[854,23] := 959.0618;
   DATA[854,24] := 2.0;
   DATA[854,25] := 2.0;
   DATA[854,26] := 7.878942;
   DATA[854,27] := 144.6039;
   DATA[854,28] := 263.0415;
   DATA[854,29] := 12.07383;
   DATA[854,30] := 1.727506;
   DATA[854,31] := 1.244012;
   DATA[854,32] := 0.7352687;
   DATA[854,33] := 0.3065689;
   DATA[854,34] := 2.0;
   DATA[854,35] := 250.8171;
   DATA[854,36] := 1.730048;
   DATA[854,37] := 189.5347;
   DATA[854,38] := 0.000128152;
   DATA[854,39] := 1.0;
   DATA[855,0] := 2.555488;
   DATA[855,1] := 586.5932;
   DATA[855,2] := 2.0;
   DATA[855,3] := 1.0;
   DATA[855,4] := 262.3366;
   DATA[855,5] := 8.460203;
   DATA[855,6] := 315.1243;
   DATA[855,8] := 1.0;
   DATA[855,9] := 1.0;
   DATA[855,10] := 1.0;
   DATA[855,11] := 2.026378;
   DATA[855,13] := 1011.359;
   DATA[855,14] := 1.0;
   DATA[855,15] := 1.0;
   DATA[855,16] := 1.0;
   DATA[855,17] := 1.0;
   DATA[855,18] := 1.0;
   DATA[855,19] := 1.0;
   DATA[855,20] := 148.808;
   DATA[855,21] := 155.3448;
   DATA[855,22] := 1.717361;
   DATA[855,23] := 958.3696;
   DATA[855,24] := 2.0;
   DATA[855,25] := 2.0;
   DATA[855,26] := 7.878942;
   DATA[855,27] := 144.6039;
   DATA[855,28] := 263.0415;
   DATA[855,29] := 12.07383;
   DATA[855,30] := 1.727506;
   DATA[855,31] := 1.243884;
   DATA[855,32] := 0.736421;
   DATA[855,33] := 0.3082983;
   DATA[855,34] := 2.0;
   DATA[855,35] := 250.8652;
   DATA[855,36] := 1.730048;
   DATA[855,37] := 189.5347;
   DATA[855,38] := 0.000128152;
   DATA[855,39] := 1.0;
   DATA[856,0] := 2.555488;
   DATA[856,1] := 587.2997;
   DATA[856,2] := 2.0;
   DATA[856,3] := 1.0;
   DATA[856,4] := 262.3366;
   DATA[856,5] := 8.460203;
   DATA[856,6] := 315.1243;
   DATA[856,8] := 1.0;
   DATA[856,9] := 1.0;
   DATA[856,10] := 1.0;
   DATA[856,11] := 2.026378;
   DATA[856,13] := 1010.879;
   DATA[856,14] := 1.0;
   DATA[856,15] := 1.0;
   DATA[856,16] := 1.0;
   DATA[856,17] := 1.0;
   DATA[856,18] := 1.0;
   DATA[856,19] := 1.0;
   DATA[856,20] := 148.808;
   DATA[856,21] := 155.3448;
   DATA[856,22] := 1.717361;
   DATA[856,23] := 957.9851;
   DATA[856,24] := 2.0;
   DATA[856,25] := 2.0;
   DATA[856,26] := 7.878942;
   DATA[856,27] := 144.6039;
   DATA[856,28] := 263.0415;
   DATA[856,29] := 12.07383;
   DATA[856,30] := 1.727506;
   DATA[856,31] := 1.258742;
   DATA[856,32] := 0.736421;
   DATA[856,33] := 0.3082983;
   DATA[856,34] := 2.0;
   DATA[856,35] := 250.8652;
   DATA[856,36] := 1.826162;
   DATA[856,37] := 189.5347;
   DATA[856,38] := 0.000128152;
   DATA[856,39] := 1.0;
   DATA[857,0] := 2.555488;
   DATA[857,1] := 587.8885;
   DATA[857,2] := 2.0;
   DATA[857,3] := 1.0;
   DATA[857,4] := 262.3366;
   DATA[857,5] := 8.460203;
   DATA[857,6] := 315.1243;
   DATA[857,8] := 1.0;
   DATA[857,9] := 1.0;
   DATA[857,10] := 1.0;
   DATA[857,11] := 2.026378;
   DATA[857,13] := 1011.239;
   DATA[857,14] := 1.0;
   DATA[857,15] := 1.0;
   DATA[857,16] := 1.0;
   DATA[857,17] := 1.0;
   DATA[857,18] := 1.0;
   DATA[857,19] := 1.0;
   DATA[857,20] := 148.808;
   DATA[857,21] := 155.3448;
   DATA[857,22] := 1.717361;
   DATA[857,23] := 957.6775;
   DATA[857,24] := 2.0;
   DATA[857,25] := 2.0;
   DATA[857,26] := 7.878942;
   DATA[857,27] := 144.8347;
   DATA[857,28] := 263.0415;
   DATA[857,29] := 12.07383;
   DATA[857,30] := 1.727506;
   DATA[857,31] := 1.269502;
   DATA[857,32] := 0.7357808;
   DATA[857,33] := 0.3068891;
   DATA[857,34] := 2.0;
   DATA[857,35] := 250.9613;
   DATA[857,36] := 1.826162;
   DATA[857,37] := 189.5347;
   DATA[857,38] := 0.000128152;
   DATA[857,39] := 1.0;
   DATA[858,0] := 2.555488;
   DATA[858,1] := 588.0456;
   DATA[858,2] := 2.0;
   DATA[858,3] := 1.0;
   DATA[858,4] := 262.3366;
   DATA[858,5] := 8.460203;
   DATA[858,6] := 315.1243;
   DATA[858,8] := 1.0;
   DATA[858,9] := 1.0;
   DATA[858,10] := 1.0;
   DATA[858,11] := 2.026378;
   DATA[858,13] := 1011.119;
   DATA[858,14] := 1.0;
   DATA[858,15] := 1.0;
   DATA[858,16] := 1.0;
   DATA[858,17] := 1.0;
   DATA[858,18] := 1.0;
   DATA[858,19] := 1.0;
   DATA[858,20] := 148.808;
   DATA[858,21] := 155.3448;
   DATA[858,22] := 1.717361;
   DATA[858,23] := 957.3699;
   DATA[858,24] := 2.0;
   DATA[858,25] := 2.0;
   DATA[858,26] := 7.878942;
   DATA[858,27] := 144.8347;
   DATA[858,28] := 263.0415;
   DATA[858,29] := 12.07383;
   DATA[858,30] := 1.727506;
   DATA[858,31] := 1.291918;
   DATA[858,32] := 0.7357808;
   DATA[858,33] := 0.3065689;
   DATA[858,34] := 2.0;
   DATA[858,35] := 250.9613;
   DATA[858,36] := 1.826162;
   DATA[858,37] := 189.6469;
   DATA[858,38] := 0.000128152;
   DATA[858,39] := 1.0;
   DATA[859,0] := 2.551645;
   DATA[859,1] := 588.0848;
   DATA[859,2] := 2.0;
   DATA[859,3] := 1.0;
   DATA[859,4] := 262.3366;
   DATA[859,5] := 8.460203;
   DATA[859,6] := 315.1243;
   DATA[859,8] := 1.0;
   DATA[859,9] := 1.0;
   DATA[859,10] := 1.0;
   DATA[859,11] := 2.026378;
   DATA[859,13] := 1011.079;
   DATA[859,14] := 1.0;
   DATA[859,15] := 1.0;
   DATA[859,16] := 1.0;
   DATA[859,17] := 1.0;
   DATA[859,18] := 1.0;
   DATA[859,19] := 1.0;
   DATA[859,20] := 148.808;
   DATA[859,21] := 155.3448;
   DATA[859,22] := 1.717361;
   DATA[859,23] := 957.3699;
   DATA[859,24] := 2.0;
   DATA[859,25] := 2.0;
   DATA[859,26] := 7.878942;
   DATA[859,27] := 144.8347;
   DATA[859,28] := 263.0415;
   DATA[859,29] := 12.07383;
   DATA[859,30] := 1.727506;
   DATA[859,31] := 1.301652;
   DATA[859,32] := 0.7353967;
   DATA[859,33] := 0.3065689;
   DATA[859,34] := 2.0;
   DATA[859,35] := 250.9613;
   DATA[859,36] := 1.826162;
   DATA[859,37] := 189.6469;
   DATA[859,38] := 0.000128152;
   DATA[859,39] := 1.0;
   DATA[860,0] := 2.542356;
   DATA[860,1] := 588.8306;
   DATA[860,2] := 2.0;
   DATA[860,3] := 1.0;
   DATA[860,4] := 262.3366;
   DATA[860,5] := 8.460203;
   DATA[860,6] := 315.1243;
   DATA[860,8] := 1.0;
   DATA[860,9] := 1.0;
   DATA[860,10] := 1.0;
   DATA[860,11] := 2.026378;
   DATA[860,13] := 1010.879;
   DATA[860,14] := 1.0;
   DATA[860,15] := 1.0;
   DATA[860,16] := 1.0;
   DATA[860,17] := 1.0;
   DATA[860,18] := 1.0;
   DATA[860,19] := 1.0;
   DATA[860,20] := 148.808;
   DATA[860,21] := 155.3448;
   DATA[860,22] := 1.717874;
   DATA[860,23] := 956.8316;
   DATA[860,24] := 2.0;
   DATA[860,25] := 2.0;
   DATA[860,26] := 7.878942;
   DATA[860,27] := 144.8347;
   DATA[860,28] := 263.0415;
   DATA[860,29] := 12.07383;
   DATA[860,30] := 1.727506;
   DATA[860,31] := 1.301652;
   DATA[860,32] := 0.7353967;
   DATA[860,33] := 0.3065689;
   DATA[860,34] := 2.0;
   DATA[860,35] := 250.9613;
   DATA[860,36] := 1.826162;
   DATA[860,37] := 189.6629;
   DATA[860,38] := 0.000128152;
   DATA[860,39] := 1.0;
   DATA[861,0] := 2.539154;
   DATA[861,1] := 589.1839;
   DATA[861,2] := 2.0;
   DATA[861,3] := 1.0;
   DATA[861,4] := 262.3366;
   DATA[861,5] := 8.460203;
   DATA[861,6] := 315.1243;
   DATA[861,8] := 1.0;
   DATA[861,9] := 1.0;
   DATA[861,10] := 1.0;
   DATA[861,11] := 2.026378;
   DATA[861,13] := 1010.959;
   DATA[861,14] := 1.0;
   DATA[861,15] := 1.0;
   DATA[861,16] := 1.0;
   DATA[861,17] := 1.0;
   DATA[861,18] := 1.0;
   DATA[861,19] := 1.0;
   DATA[861,20] := 148.808;
   DATA[861,21] := 155.3448;
   DATA[861,22] := 1.717874;
   DATA[861,23] := 956.4855;
   DATA[861,24] := 2.0;
   DATA[861,25] := 2.0;
   DATA[861,26] := 7.878942;
   DATA[861,27] := 144.8347;
   DATA[861,28] := 263.0415;
   DATA[861,29] := 12.07383;
   DATA[861,30] := 1.729813;
   DATA[861,31] := 1.285129;
   DATA[861,32] := 0.7353967;
   DATA[861,33] := 0.3065689;
   DATA[861,34] := 2.0;
   DATA[861,35] := 250.9613;
   DATA[861,36] := 1.746067;
   DATA[861,37] := 189.6629;
   DATA[861,38] := 0.000128152;
   DATA[861,39] := 1.0;
   DATA[862,0] := 2.53435;
   DATA[862,1] := 589.7335;
   DATA[862,2] := 2.0;
   DATA[862,3] := 1.0;
   DATA[862,4] := 262.3366;
   DATA[862,5] := 8.460203;
   DATA[862,6] := 315.1243;
   DATA[862,8] := 1.0;
   DATA[862,9] := 1.0;
   DATA[862,10] := 1.0;
   DATA[862,11] := 2.026378;
   DATA[862,13] := 1010.718;
   DATA[862,14] := 1.0;
   DATA[862,15] := 1.0;
   DATA[862,16] := 1.0;
   DATA[862,17] := 1.0;
   DATA[862,18] := 1.0;
   DATA[862,19] := 1.0;
   DATA[862,20] := 148.808;
   DATA[862,21] := 155.3448;
   DATA[862,22] := 1.717874;
   DATA[862,23] := 956.0626;
   DATA[862,24] := 2.0;
   DATA[862,25] := 2.0;
   DATA[862,26] := 7.878942;
   DATA[862,27] := 144.7321;
   DATA[862,28] := 263.0415;
   DATA[862,29] := 12.07383;
   DATA[862,30] := 1.729813;
   DATA[862,31] := 1.273473;
   DATA[862,32] := 0.7353967;
   DATA[862,33] := 0.3065689;
   DATA[862,34] := 2.0;
   DATA[862,35] := 250.9613;
   DATA[862,36] := 1.746067;
   DATA[862,37] := 189.6629;
   DATA[862,38] := 0.000128152;
   DATA[862,39] := 1.0;
   DATA[863,0] := 2.53435;
   DATA[863,1] := 590.1652;
   DATA[863,2] := 2.0;
   DATA[863,3] := 1.0;
   DATA[863,4] := 262.3366;
   DATA[863,5] := 8.460203;
   DATA[863,6] := 315.1243;
   DATA[863,8] := 1.0;
   DATA[863,9] := 1.0;
   DATA[863,10] := 1.0;
   DATA[863,11] := 2.026378;
   DATA[863,13] := 1010.518;
   DATA[863,14] := 1.0;
   DATA[863,15] := 1.0;
   DATA[863,16] := 1.0;
   DATA[863,17] := 1.0;
   DATA[863,18] := 1.0;
   DATA[863,19] := 1.0;
   DATA[863,20] := 148.808;
   DATA[863,21] := 155.3448;
   DATA[863,22] := 1.717874;
   DATA[863,23] := 955.4473;
   DATA[863,24] := 2.0;
   DATA[863,25] := 2.0;
   DATA[863,26] := 7.878942;
   DATA[863,27] := 144.7321;
   DATA[863,28] := 263.0415;
   DATA[863,29] := 12.07383;
   DATA[863,30] := 1.729813;
   DATA[863,31] := 1.271935;
   DATA[863,32] := 0.7353967;
   DATA[863,33] := 0.3065689;
   DATA[863,34] := 2.0;
   DATA[863,35] := 250.9613;
   DATA[863,36] := 1.746067;
   DATA[863,37] := 189.6629;
   DATA[863,38] := 0.000128152;
   DATA[863,39] := 1.0;
   DATA[864,0] := 2.543638;
   DATA[864,1] := 590.911;
   DATA[864,2] := 2.0;
   DATA[864,3] := 1.0;
   DATA[864,4] := 262.3366;
   DATA[864,5] := 8.460203;
   DATA[864,6] := 315.1243;
   DATA[864,8] := 1.0;
   DATA[864,9] := 1.0;
   DATA[864,10] := 1.0;
   DATA[864,11] := 2.026378;
   DATA[864,13] := 1011.319;
   DATA[864,14] := 1.0;
   DATA[864,15] := 1.0;
   DATA[864,16] := 1.0;
   DATA[864,17] := 1.0;
   DATA[864,18] := 1.0;
   DATA[864,19] := 1.0;
   DATA[864,20] := 148.808;
   DATA[864,21] := 155.3448;
   DATA[864,22] := 1.717874;
   DATA[864,23] := 955.1782;
   DATA[864,24] := 2.0;
   DATA[864,25] := 2.0;
   DATA[864,26] := 7.878942;
   DATA[864,27] := 144.7065;
   DATA[864,28] := 263.0415;
   DATA[864,29] := 12.07383;
   DATA[864,30] := 1.729813;
   DATA[864,31] := 1.289868;
   DATA[864,32] := 0.7353967;
   DATA[864,33] := 0.3065689;
   DATA[864,34] := 2.0;
   DATA[864,35] := 250.9613;
   DATA[864,36] := 1.746067;
   DATA[864,37] := 189.6629;
   DATA[864,38] := 0.000128152;
   DATA[864,39] := 1.0;
   DATA[865,0] := 2.553886;
   DATA[865,1] := 591.7746;
   DATA[865,2] := 2.0;
   DATA[865,3] := 1.0;
   DATA[865,4] := 262.3366;
   DATA[865,5] := 8.460203;
   DATA[865,6] := 315.1243;
   DATA[865,8] := 1.0;
   DATA[865,9] := 1.0;
   DATA[865,10] := 1.0;
   DATA[865,11] := 2.026378;
   DATA[865,13] := 1011.039;
   DATA[865,14] := 1.0;
   DATA[865,15] := 1.0;
   DATA[865,16] := 1.0;
   DATA[865,17] := 1.0;
   DATA[865,18] := 1.0;
   DATA[865,19] := 1.0;
   DATA[865,20] := 148.808;
   DATA[865,21] := 155.5499;
   DATA[865,22] := 1.717874;
   DATA[865,23] := 954.9859;
   DATA[865,24] := 2.0;
   DATA[865,25] := 2.0;
   DATA[865,26] := 7.878942;
   DATA[865,27] := 144.7065;
   DATA[865,28] := 263.0415;
   DATA[865,29] := 12.07383;
   DATA[865,30] := 1.729813;
   DATA[865,31] := 1.301396;
   DATA[865,32] := 0.7353967;
   DATA[865,33] := 0.3065689;
   DATA[865,34] := 2.0;
   DATA[865,35] := 250.9453;
   DATA[865,36] := 1.746067;
   DATA[865,37] := 189.6629;
   DATA[865,38] := 0.000128152;
   DATA[865,39] := 1.0;
   DATA[866,0] := 2.558691;
   DATA[866,1] := 592.7952;
   DATA[866,2] := 2.0;
   DATA[866,3] := 1.0;
   DATA[866,4] := 262.3366;
   DATA[866,5] := 8.460203;
   DATA[866,6] := 315.1243;
   DATA[866,8] := 1.0;
   DATA[866,9] := 1.0;
   DATA[866,10] := 1.0;
   DATA[866,11] := 2.026378;
   DATA[866,13] := 1011.039;
   DATA[866,14] := 1.0;
   DATA[866,15] := 1.0;
   DATA[866,16] := 1.0;
   DATA[866,17] := 1.0;
   DATA[866,18] := 1.0;
   DATA[866,19] := 1.0;
   DATA[866,20] := 148.808;
   DATA[866,21] := 155.5499;
   DATA[866,22] := 1.717874;
   DATA[866,23] := 954.8705;
   DATA[866,24] := 2.0;
   DATA[866,25] := 2.0;
   DATA[866,26] := 7.878942;
   DATA[866,27] := 144.7065;
   DATA[866,28] := 263.0415;
   DATA[866,29] := 12.07383;
   DATA[866,30] := 1.729813;
   DATA[866,31] := 1.310106;
   DATA[866,32] := 0.7353967;
   DATA[866,33] := 0.3065689;
   DATA[866,34] := 2.0;
   DATA[866,35] := 250.8652;
   DATA[866,36] := 1.746067;
   DATA[866,37] := 189.6629;
   DATA[866,38] := 0.000128152;
   DATA[866,39] := 1.0;
   DATA[867,0] := 2.558691;
   DATA[867,1] := 593.6587;
   DATA[867,2] := 2.0;
   DATA[867,3] := 1.0;
   DATA[867,4] := 262.3366;
   DATA[867,5] := 8.460203;
   DATA[867,6] := 315.1243;
   DATA[867,8] := 1.0;
   DATA[867,9] := 1.0;
   DATA[867,10] := 1.0;
   DATA[867,11] := 2.026378;
   DATA[867,13] := 1011.64;
   DATA[867,14] := 1.0;
   DATA[867,15] := 1.0;
   DATA[867,16] := 1.0;
   DATA[867,17] := 1.0;
   DATA[867,18] := 1.0;
   DATA[867,19] := 1.0;
   DATA[867,20] := 148.808;
   DATA[867,21] := 155.5499;
   DATA[867,22] := 1.717874;
   DATA[867,23] := 954.3322;
   DATA[867,24] := 2.0;
   DATA[867,25] := 2.0;
   DATA[867,26] := 7.878942;
   DATA[867,27] := 144.7065;
   DATA[867,28] := 263.0415;
   DATA[867,29] := 12.07383;
   DATA[867,30] := 1.7293;
   DATA[867,31] := 1.312284;
   DATA[867,32] := 0.7353967;
   DATA[867,33] := 0.3065689;
   DATA[867,34] := 2.0;
   DATA[867,35] := 250.8652;
   DATA[867,36] := 1.746067;
   DATA[867,37] := 189.6629;
   DATA[867,38] := 0.000128152;
   DATA[867,39] := 1.0;
   DATA[868,0] := 2.563495;
   DATA[868,1] := 594.3652;
   DATA[868,2] := 2.0;
   DATA[868,3] := 1.0;
   DATA[868,4] := 262.3366;
   DATA[868,5] := 8.460203;
   DATA[868,6] := 315.1243;
   DATA[868,8] := 1.0;
   DATA[868,9] := 1.0;
   DATA[868,10] := 1.0;
   DATA[868,11] := 2.026378;
   DATA[868,13] := 1011.52;
   DATA[868,14] := 1.0;
   DATA[868,15] := 1.0;
   DATA[868,16] := 1.0;
   DATA[868,17] := 1.0;
   DATA[868,18] := 1.0;
   DATA[868,19] := 1.0;
   DATA[868,20] := 148.808;
   DATA[868,21] := 155.5499;
   DATA[868,22] := 1.717874;
   DATA[868,23] := 954.1015;
   DATA[868,24] := 2.0;
   DATA[868,25] := 2.0;
   DATA[868,26] := 7.878942;
   DATA[868,27] := 144.7065;
   DATA[868,28] := 263.0415;
   DATA[868,29] := 12.07383;
   DATA[868,30] := 1.726737;
   DATA[868,31] := 1.312284;
   DATA[868,32] := 0.7353967;
   DATA[868,33] := 0.3065689;
   DATA[868,34] := 2.0;
   DATA[868,35] := 250.785;
   DATA[868,36] := 1.746067;
   DATA[868,37] := 189.4546;
   DATA[868,38] := 0.000128152;
   DATA[868,39] := 1.0;
   DATA[869,0] := 2.565737;
   DATA[869,1] := 595.0325;
   DATA[869,2] := 2.0;
   DATA[869,3] := 1.0;
   DATA[869,4] := 262.3366;
   DATA[869,5] := 8.460203;
   DATA[869,6] := 315.1243;
   DATA[869,8] := 1.0;
   DATA[869,9] := 1.0;
   DATA[869,10] := 1.0;
   DATA[869,11] := 2.026378;
   DATA[869,13] := 1011.479;
   DATA[869,14] := 1.0;
   DATA[869,15] := 1.0;
   DATA[869,16] := 1.0;
   DATA[869,17] := 1.0;
   DATA[869,18] := 1.0;
   DATA[869,19] := 1.0;
   DATA[869,20] := 148.808;
   DATA[869,21] := 155.5499;
   DATA[869,22] := 1.717874;
   DATA[869,23] := 953.7939;
   DATA[869,24] := 2.0;
   DATA[869,25] := 2.0;
   DATA[869,26] := 7.878942;
   DATA[869,27] := 144.7065;
   DATA[869,28] := 263.0415;
   DATA[869,29] := 12.07383;
   DATA[869,30] := 1.726096;
   DATA[869,31] := 1.302165;
   DATA[869,32] := 0.7353967;
   DATA[869,33] := 0.3072735;
   DATA[869,34] := 2.0;
   DATA[869,35] := 250.6409;
   DATA[869,36] := 1.746067;
   DATA[869,37] := 189.3745;
   DATA[869,38] := 0.000128152;
   DATA[869,39] := 1.0;
   DATA[870,0] := 2.565737;
   DATA[870,1] := 595.8176;
   DATA[870,2] := 2.0;
   DATA[870,3] := 1.0;
   DATA[870,4] := 262.3366;
   DATA[870,5] := 8.460203;
   DATA[870,6] := 315.1243;
   DATA[870,8] := 1.0;
   DATA[870,9] := 1.0;
   DATA[870,10] := 1.0;
   DATA[870,11] := 2.026378;
   DATA[870,13] := 1010.919;
   DATA[870,14] := 1.0;
   DATA[870,15] := 1.0;
   DATA[870,16] := 1.0;
   DATA[870,17] := 1.0;
   DATA[870,18] := 1.0;
   DATA[870,19] := 1.0;
   DATA[870,20] := 148.808;
   DATA[870,21] := 155.5499;
   DATA[870,22] := 1.716849;
   DATA[870,23] := 953.3325;
   DATA[870,24] := 2.0;
   DATA[870,25] := 2.0;
   DATA[870,26] := 7.878942;
   DATA[870,27] := 144.7065;
   DATA[870,28] := 263.0415;
   DATA[870,29] := 12.07383;
   DATA[870,30] := 1.726096;
   DATA[870,31] := 1.302165;
   DATA[870,32] := 0.7353967;
   DATA[870,33] := 0.3083624;
   DATA[870,34] := 2.0;
   DATA[870,35] := 250.5768;
   DATA[870,36] := 1.746067;
   DATA[870,37] := 189.3425;
   DATA[870,38] := 0.000128152;
   DATA[870,39] := 1.0;
   DATA[871,0] := 2.555168;
   DATA[871,1] := 596.3279;
   DATA[871,2] := 2.0;
   DATA[871,3] := 1.0;
   DATA[871,4] := 262.3366;
   DATA[871,5] := 8.460844;
   DATA[871,6] := 315.1243;
   DATA[871,8] := 1.0;
   DATA[871,9] := 1.0;
   DATA[871,10] := 1.0;
   DATA[871,11] := 2.026378;
   DATA[871,13] := 1011.319;
   DATA[871,14] := 1.0;
   DATA[871,15] := 1.0;
   DATA[871,16] := 1.0;
   DATA[871,17] := 1.0;
   DATA[871,18] := 1.0;
   DATA[871,19] := 1.0;
   DATA[871,20] := 148.808;
   DATA[871,21] := 155.4473;
   DATA[871,22] := 1.716721;
   DATA[871,23] := 952.8326;
   DATA[871,24] := 2.0;
   DATA[871,25] := 2.0;
   DATA[871,26] := 7.878942;
   DATA[871,27] := 144.7065;
   DATA[871,28] := 263.0415;
   DATA[871,29] := 12.07383;
   DATA[871,30] := 1.726096;
   DATA[871,31] := 1.302165;
   DATA[871,32] := 0.7379573;
   DATA[871,33] := 0.3083624;
   DATA[871,34] := 2.0;
   DATA[871,35] := 250.4967;
   DATA[871,36] := 1.746067;
   DATA[871,37] := 189.2143;
   DATA[871,38] := 0.000128152;
   DATA[871,39] := 1.0;
   DATA[872,0] := 2.551965;
   DATA[872,1] := 596.6812;
   DATA[872,2] := 2.0;
   DATA[872,3] := 1.0;
   DATA[872,4] := 262.3366;
   DATA[872,5] := 8.462126;
   DATA[872,6] := 315.1243;
   DATA[872,8] := 1.0;
   DATA[872,9] := 1.0;
   DATA[872,10] := 1.0;
   DATA[872,11] := 2.010372;
   DATA[872,13] := 1011.079;
   DATA[872,14] := 1.0;
   DATA[872,15] := 1.0;
   DATA[872,16] := 1.0;
   DATA[872,17] := 1.0;
   DATA[872,18] := 1.0;
   DATA[872,19] := 1.0;
   DATA[872,20] := 148.808;
   DATA[872,21] := 155.4473;
   DATA[872,22] := 1.71467;
   DATA[872,23] := 952.6788;
   DATA[872,24] := 2.0;
   DATA[872,25] := 2.0;
   DATA[872,26] := 7.878942;
   DATA[872,27] := 144.7065;
   DATA[872,28] := 263.0415;
   DATA[872,29] := 12.07383;
   DATA[872,30] := 1.726096;
   DATA[872,31] := 1.293711;
   DATA[872,32] := 0.7379573;
   DATA[872,33] := 0.3083624;
   DATA[872,34] := 2.0;
   DATA[872,35] := 250.2724;
   DATA[872,36] := 1.746067;
   DATA[872,37] := 189.1983;
   DATA[872,38] := 0.000128152;
   DATA[872,39] := 1.0;
   DATA[873,0] := 2.548121;
   DATA[873,1] := 596.7204;
   DATA[873,2] := 2.0;
   DATA[873,3] := 1.0;
   DATA[873,4] := 262.3366;
   DATA[873,5] := 8.462126;
   DATA[873,6] := 315.1243;
   DATA[873,8] := 1.0;
   DATA[873,9] := 1.0;
   DATA[873,10] := 1.0;
   DATA[873,11] := 2.010372;
   DATA[873,13] := 1011.119;
   DATA[873,14] := 1.0;
   DATA[873,15] := 1.0;
   DATA[873,16] := 1.0;
   DATA[873,17] := 1.0;
   DATA[873,18] := 1.0;
   DATA[873,19] := 1.0;
   DATA[873,20] := 148.808;
   DATA[873,21] := 155.4473;
   DATA[873,22] := 1.714286;
   DATA[873,23] := 952.6019;
   DATA[873,24] := 2.0;
   DATA[873,25] := 2.0;
   DATA[873,26] := 7.878942;
   DATA[873,27] := 144.7065;
   DATA[873,28] := 263.0415;
   DATA[873,29] := 12.07383;
   DATA[873,30] := 1.726096;
   DATA[873,31] := 1.291789;
   DATA[873,32] := 0.7379573;
   DATA[873,33] := 0.3083624;
   DATA[873,34] := 2.0;
   DATA[873,35] := 250.2724;
   DATA[873,36] := 1.746067;
   DATA[873,37] := 189.022;
   DATA[873,38] := 0.000128152;
   DATA[873,39] := 1.0;
   DATA[874,0] := 2.548121;
   DATA[874,1] := 596.6419;
   DATA[874,2] := 2.0;
   DATA[874,3] := 1.0;
   DATA[874,4] := 262.3366;
   DATA[874,5] := 8.462126;
   DATA[874,6] := 315.1243;
   DATA[874,8] := 1.0;
   DATA[874,9] := 1.0;
   DATA[874,10] := 1.0;
   DATA[874,11] := 2.010372;
   DATA[874,13] := 1010.839;
   DATA[874,14] := 1.0;
   DATA[874,15] := 1.0;
   DATA[874,16] := 1.0;
   DATA[874,17] := 1.0;
   DATA[874,18] := 1.0;
   DATA[874,19] := 1.0;
   DATA[874,20] := 148.808;
   DATA[874,21] := 155.4473;
   DATA[874,22] := 1.714286;
   DATA[874,23] := 952.1021;
   DATA[874,24] := 2.0;
   DATA[874,25] := 2.0;
   DATA[874,26] := 7.878942;
   DATA[874,27] := 144.7065;
   DATA[874,28] := 263.0415;
   DATA[874,29] := 12.07383;
   DATA[874,30] := 1.726096;
   DATA[874,31] := 1.28372;
   DATA[874,32] := 0.7379573;
   DATA[874,33] := 0.3083624;
   DATA[874,34] := 2.0;
   DATA[874,35] := 250.1762;
   DATA[874,36] := 1.746067;
   DATA[874,37] := 189.022;
   DATA[874,38] := 0.000128152;
   DATA[874,39] := 1.0;
   DATA[875,0] := 2.548121;
   DATA[875,1] := 597.0344;
   DATA[875,2] := 2.0;
   DATA[875,3] := 1.0;
   DATA[875,4] := 262.3366;
   DATA[875,5] := 8.462126;
   DATA[875,6] := 315.1243;
   DATA[875,8] := 1.0;
   DATA[875,9] := 1.0;
   DATA[875,10] := 1.0;
   DATA[875,11] := 2.010372;
   DATA[875,13] := 1011.119;
   DATA[875,14] := 1.0;
   DATA[875,15] := 1.0;
   DATA[875,16] := 1.0;
   DATA[875,17] := 1.0;
   DATA[875,18] := 1.0;
   DATA[875,19] := 1.0;
   DATA[875,20] := 148.808;
   DATA[875,21] := 155.4473;
   DATA[875,22] := 1.713261;
   DATA[875,23] := 951.4099;
   DATA[875,24] := 2.0;
   DATA[875,25] := 2.0;
   DATA[875,26] := 7.878942;
   DATA[875,27] := 144.7065;
   DATA[875,28] := 263.0415;
   DATA[875,29] := 12.07383;
   DATA[875,30] := 1.726096;
   DATA[875,31] := 1.281927;
   DATA[875,32] := 0.7347566;
   DATA[875,33] := 0.3083624;
   DATA[875,34] := 2.0;
   DATA[875,35] := 250.1762;
   DATA[875,36] := 1.746067;
   DATA[875,37] := 189.022;
   DATA[875,38] := 0.000128152;
   DATA[875,39] := 1.0;
   DATA[876,0] := 2.553886;
   DATA[876,1] := 596.8774;
   DATA[876,2] := 2.0;
   DATA[876,3] := 1.0;
   DATA[876,4] := 262.3366;
   DATA[876,5] := 8.462126;
   DATA[876,6] := 315.1243;
   DATA[876,8] := 1.0;
   DATA[876,9] := 1.0;
   DATA[876,10] := 1.0;
   DATA[876,11] := 2.032781;
   DATA[876,13] := 1011.079;
   DATA[876,14] := 1.0;
   DATA[876,15] := 1.0;
   DATA[876,16] := 1.0;
   DATA[876,17] := 1.0;
   DATA[876,18] := 1.0;
   DATA[876,19] := 1.0;
   DATA[876,20] := 148.808;
   DATA[876,21] := 155.4473;
   DATA[876,22] := 1.713261;
   DATA[876,23] := 951.1023;
   DATA[876,24] := 2.0;
   DATA[876,25] := 2.0;
   DATA[876,26] := 7.878942;
   DATA[876,27] := 144.7065;
   DATA[876,28] := 263.0415;
   DATA[876,29] := 12.07383;
   DATA[876,30] := 1.726096;
   DATA[876,31] := 1.281286;
   DATA[876,32] := 0.7347566;
   DATA[876,33] := 0.3083624;
   DATA[876,34] := 2.0;
   DATA[876,35] := 250.1762;
   DATA[876,36] := 1.746067;
   DATA[876,37] := 189.022;
   DATA[876,38] := 0.000128152;
   DATA[876,39] := 1.0;
   DATA[877,0] := 2.553886;
   DATA[877,1] := 596.6812;
   DATA[877,2] := 2.0;
   DATA[877,3] := 1.0;
   DATA[877,4] := 262.3366;
   DATA[877,5] := 8.462126;
   DATA[877,6] := 315.1243;
   DATA[877,8] := 1.0;
   DATA[877,9] := 1.0;
   DATA[877,10] := 1.0;
   DATA[877,11] := 2.032781;
   DATA[877,13] := 1011.159;
   DATA[877,14] := 1.0;
   DATA[877,15] := 1.0;
   DATA[877,16] := 1.0;
   DATA[877,17] := 1.0;
   DATA[877,18] := 1.0;
   DATA[877,19] := 1.0;
   DATA[877,20] := 148.808;
   DATA[877,21] := 155.4473;
   DATA[877,22] := 1.713261;
   DATA[877,23] := 951.0254;
   DATA[877,24] := 2.0;
   DATA[877,25] := 2.0;
   DATA[877,26] := 7.878942;
   DATA[877,27] := 144.7065;
   DATA[877,28] := 263.0415;
   DATA[877,29] := 12.07383;
   DATA[877,30] := 1.726096;
   DATA[877,31] := 1.274113;
   DATA[877,32] := 0.7347566;
   DATA[877,33] := 0.3065689;
   DATA[877,34] := 2.0;
   DATA[877,35] := 250.3525;
   DATA[877,36] := 1.746067;
   DATA[877,37] := 189.1342;
   DATA[877,38] := 0.000128152;
   DATA[877,39] := 1.0;
   DATA[878,0] := 2.553886;
   DATA[878,1] := 596.9167;
   DATA[878,2] := 2.0;
   DATA[878,3] := 1.0;
   DATA[878,4] := 262.3686;
   DATA[878,5] := 8.462126;
   DATA[878,6] := 315.1243;
   DATA[878,8] := 1.0;
   DATA[878,9] := 1.0;
   DATA[878,10] := 1.0;
   DATA[878,11] := 2.032781;
   DATA[878,13] := 1010.758;
   DATA[878,14] := 1.0;
   DATA[878,15] := 1.0;
   DATA[878,16] := 1.0;
   DATA[878,17] := 1.0;
   DATA[878,18] := 1.0;
   DATA[878,19] := 1.0;
   DATA[878,20] := 148.808;
   DATA[878,21] := 155.4473;
   DATA[878,22] := 1.714542;
   DATA[878,23] := 951.0254;
   DATA[878,24] := 2.0;
   DATA[878,25] := 2.0;
   DATA[878,26] := 7.878942;
   DATA[878,27] := 144.7065;
   DATA[878,28] := 263.0415;
   DATA[878,29] := 12.07383;
   DATA[878,30] := 1.726096;
   DATA[878,31] := 1.27232;
   DATA[878,32] := 0.7347566;
   DATA[878,33] := 0.3065689;
   DATA[878,34] := 2.0;
   DATA[878,35] := 250.3845;
   DATA[878,36] := 1.746067;
   DATA[878,37] := 189.2784;
   DATA[878,38] := 0.000128152;
   DATA[878,39] := 1.0;
   DATA[879,0] := 2.553886;
   DATA[879,1] := 597.2307;
   DATA[879,2] := 2.0;
   DATA[879,3] := 1.0;
   DATA[879,4] := 262.3686;
   DATA[879,5] := 8.462126;
   DATA[879,6] := 315.1243;
   DATA[879,8] := 1.0;
   DATA[879,9] := 1.0;
   DATA[879,10] := 1.0;
   DATA[879,11] := 2.032781;
   DATA[879,13] := 1010.839;
   DATA[879,14] := 1.0;
   DATA[879,15] := 1.0;
   DATA[879,16] := 1.0;
   DATA[879,17] := 1.0;
   DATA[879,18] := 1.0;
   DATA[879,19] := 1.0;
   DATA[879,20] := 148.808;
   DATA[879,21] := 155.4473;
   DATA[879,22] := 1.715311;
   DATA[879,23] := 950.4486;
   DATA[879,24] := 2.0;
   DATA[879,25] := 2.0;
   DATA[879,26] := 7.878942;
   DATA[879,27] := 144.7065;
   DATA[879,28] := 263.0415;
   DATA[879,29] := 12.07383;
   DATA[879,30] := 1.726096;
   DATA[879,31] := 1.271295;
   DATA[879,32] := 0.7353967;
   DATA[879,33] := 0.3065689;
   DATA[879,34] := 2.0;
   DATA[879,35] := 250.5928;
   DATA[879,36] := 1.746067;
   DATA[879,37] := 189.2784;
   DATA[879,38] := 0.000128152;
   DATA[879,39] := 1.0;
   DATA[880,0] := 2.548762;
   DATA[880,1] := 597.7017;
   DATA[880,2] := 2.0;
   DATA[880,3] := 1.0;
   DATA[880,4] := 262.3686;
   DATA[880,5] := 8.462126;
   DATA[880,6] := 315.1243;
   DATA[880,8] := 1.0;
   DATA[880,9] := 1.0;
   DATA[880,10] := 1.0;
   DATA[880,11] := 2.032781;
   DATA[880,13] := 1010.638;
   DATA[880,14] := 1.0;
   DATA[880,15] := 1.0;
   DATA[880,16] := 1.0;
   DATA[880,17] := 1.0;
   DATA[880,18] := 1.0;
   DATA[880,19] := 1.0;
   DATA[880,20] := 148.808;
   DATA[880,21] := 155.4473;
   DATA[880,22] := 1.717105;
   DATA[880,23] := 950.1794;
   DATA[880,24] := 2.0;
   DATA[880,25] := 2.0;
   DATA[880,26] := 7.878942;
   DATA[880,27] := 144.7065;
   DATA[880,28] := 263.0415;
   DATA[880,29] := 12.07383;
   DATA[880,30] := 1.726096;
   DATA[880,31] := 1.272832;
   DATA[880,32] := 0.7353967;
   DATA[880,33] := 0.3065689;
   DATA[880,34] := 2.0;
   DATA[880,35] := 250.6248;
   DATA[880,36] := 1.746067;
   DATA[880,37] := 189.2784;
   DATA[880,38] := 0.000128152;
   DATA[880,39] := 1.0;
   DATA[881,0] := 2.548121;
   DATA[881,1] := 598.2905;
   DATA[881,2] := 2.0;
   DATA[881,3] := 1.0;
   DATA[881,4] := 262.3686;
   DATA[881,5] := 8.464048;
   DATA[881,6] := 315.1243;
   DATA[881,8] := 1.0;
   DATA[881,9] := 1.0;
   DATA[881,10] := 1.0;
   DATA[881,11] := 2.026378;
   DATA[881,13] := 1010.879;
   DATA[881,14] := 1.0;
   DATA[881,15] := 1.0;
   DATA[881,16] := 1.0;
   DATA[881,17] := 1.0;
   DATA[881,18] := 1.0;
   DATA[881,19] := 1.0;
   DATA[881,20] := 148.808;
   DATA[881,21] := 155.4473;
   DATA[881,22] := 1.717746;
   DATA[881,23] := 950.1025;
   DATA[881,24] := 2.0;
   DATA[881,25] := 2.0;
   DATA[881,26] := 7.878942;
   DATA[881,27] := 144.7065;
   DATA[881,28] := 263.0415;
   DATA[881,29] := 12.07383;
   DATA[881,30] := 1.726096;
   DATA[881,31] := 1.28167;
   DATA[881,32] := 0.7353967;
   DATA[881,33] := 0.3065689;
   DATA[881,34] := 2.0;
   DATA[881,35] := 250.6248;
   DATA[881,36] := 1.746067;
   DATA[881,37] := 189.3425;
   DATA[881,38] := 0.000128152;
   DATA[881,39] := 1.0;
   DATA[882,0] := 2.543317;
   DATA[882,1] := 599.4681;
   DATA[882,2] := 2.0;
   DATA[882,3] := 1.0;
   DATA[882,4] := 262.3686;
   DATA[882,5] := 8.464048;
   DATA[882,6] := 315.1243;
   DATA[882,8] := 1.0;
   DATA[882,9] := 1.0;
   DATA[882,10] := 1.0;
   DATA[882,11] := 2.010372;
   DATA[882,13] := 1010.839;
   DATA[882,14] := 1.0;
   DATA[882,15] := 1.0;
   DATA[882,16] := 1.0;
   DATA[882,17] := 1.0;
   DATA[882,18] := 1.0;
   DATA[882,19] := 1.0;
   DATA[882,20] := 148.808;
   DATA[882,21] := 155.4473;
   DATA[882,22] := 1.717746;
   DATA[882,23] := 949.8718;
   DATA[882,24] := 2.0;
   DATA[882,25] := 2.0;
   DATA[882,26] := 7.878942;
   DATA[882,27] := 144.7065;
   DATA[882,28] := 263.0415;
   DATA[882,29] := 12.07383;
   DATA[882,30] := 1.726096;
   DATA[882,31] := 1.282439;
   DATA[882,32] := 0.7353967;
   DATA[882,33] := 0.3065689;
   DATA[882,34] := 2.0;
   DATA[882,35] := 250.6248;
   DATA[882,36] := 1.746067;
   DATA[882,37] := 189.3425;
   DATA[882,38] := 0.000128152;
   DATA[882,39] := 1.0;
   DATA[883,0] := 2.541075;
   DATA[883,1] := 600.1354;
   DATA[883,2] := 2.0;
   DATA[883,3] := 1.0;
   DATA[883,4] := 262.3686;
   DATA[883,5] := 8.464048;
   DATA[883,6] := 315.1243;
   DATA[883,8] := 1.0;
   DATA[883,9] := 1.0;
   DATA[883,10] := 1.0;
   DATA[883,11] := 2.010372;
   DATA[883,13] := 1011.319;
   DATA[883,14] := 1.0;
   DATA[883,15] := 1.0;
   DATA[883,16] := 1.0;
   DATA[883,17] := 1.0;
   DATA[883,18] := 1.0;
   DATA[883,19] := 1.0;
   DATA[883,20] := 148.808;
   DATA[883,21] := 155.4473;
   DATA[883,22] := 1.719156;
   DATA[883,23] := 949.5258;
   DATA[883,24] := 2.0;
   DATA[883,25] := 2.0;
   DATA[883,26] := 7.878942;
   DATA[883,27] := 144.7065;
   DATA[883,28] := 263.0415;
   DATA[883,29] := 12.07383;
   DATA[883,30] := 1.726096;
   DATA[883,31] := 1.276162;
   DATA[883,32] := 0.7353967;
   DATA[883,33] := 0.3065689;
   DATA[883,34] := 2.0;
   DATA[883,35] := 250.6729;
   DATA[883,36] := 1.746067;
   DATA[883,37] := 189.5187;
   DATA[883,38] := 0.000128152;
   DATA[883,39] := 1.0;
   DATA[884,0] := 2.536271;
   DATA[884,1] := 600.999;
   DATA[884,2] := 2.0;
   DATA[884,3] := 1.0;
   DATA[884,4] := 262.3686;
   DATA[884,5] := 8.464048;
   DATA[884,6] := 315.1243;
   DATA[884,8] := 1.0;
   DATA[884,9] := 1.0;
   DATA[884,10] := 1.0;
   DATA[884,11] := 2.010372;
   DATA[884,13] := 1011.079;
   DATA[884,14] := 1.0;
   DATA[884,15] := 1.0;
   DATA[884,16] := 1.0;
   DATA[884,17] := 1.0;
   DATA[884,18] := 1.0;
   DATA[884,19] := 1.0;
   DATA[884,20] := 148.808;
   DATA[884,21] := 155.4473;
   DATA[884,22] := 1.719284;
   DATA[884,23] := 949.0259;
   DATA[884,24] := 2.0;
   DATA[884,25] := 2.0;
   DATA[884,26] := 7.878942;
   DATA[884,27] := 144.5783;
   DATA[884,28] := 263.0415;
   DATA[884,29] := 12.07383;
   DATA[884,30] := 1.726352;
   DATA[884,31] := 1.262713;
   DATA[884,32] := 0.7353967;
   DATA[884,33] := 0.3065689;
   DATA[884,34] := 2.0;
   DATA[884,35] := 250.6729;
   DATA[884,36] := 1.746067;
   DATA[884,37] := 189.5187;
   DATA[884,38] := 0.000128152;
   DATA[884,39] := 1.0;
   DATA[885,0] := 2.536271;
   DATA[885,1] := 602.1373;
   DATA[885,2] := 2.0;
   DATA[885,3] := 1.0;
   DATA[885,4] := 262.3686;
   DATA[885,5] := 8.464048;
   DATA[885,6] := 315.1243;
   DATA[885,8] := 1.0;
   DATA[885,9] := 1.0;
   DATA[885,10] := 1.0;
   DATA[885,11] := 2.010372;
   DATA[885,13] := 1011.239;
   DATA[885,14] := 1.0;
   DATA[885,15] := 1.0;
   DATA[885,16] := 1.0;
   DATA[885,17] := 1.0;
   DATA[885,18] := 1.0;
   DATA[885,19] := 1.0;
   DATA[885,20] := 148.808;
   DATA[885,21] := 155.4473;
   DATA[885,22] := 1.719284;
   DATA[885,23] := 948.7183;
   DATA[885,24] := 2.0;
   DATA[885,25] := 2.0;
   DATA[885,26] := 7.878942;
   DATA[885,27] := 144.5783;
   DATA[885,28] := 263.0415;
   DATA[885,29] := 12.07383;
   DATA[885,30] := 1.726865;
   DATA[885,31] := 1.263353;
   DATA[885,32] := 0.7353967;
   DATA[885,33] := 0.3065689;
   DATA[885,34] := 2.0;
   DATA[885,35] := 250.6729;
   DATA[885,36] := 1.746067;
   DATA[885,37] := 189.5187;
   DATA[885,38] := 0.000128152;
   DATA[885,39] := 1.0;
   DATA[886,0] := 2.536271;
   DATA[886,1] := 603.0793;
   DATA[886,2] := 2.0;
   DATA[886,3] := 1.0;
   DATA[886,4] := 262.3686;
   DATA[886,5] := 8.464048;
   DATA[886,6] := 315.1243;
   DATA[886,8] := 1.0;
   DATA[886,9] := 1.0;
   DATA[886,10] := 1.0;
   DATA[886,11] := 2.010372;
   DATA[886,13] := 1010.839;
   DATA[886,14] := 1.0;
   DATA[886,15] := 1.0;
   DATA[886,16] := 1.0;
   DATA[886,17] := 1.0;
   DATA[886,18] := 1.0;
   DATA[886,19] := 1.0;
   DATA[886,20] := 148.808;
   DATA[886,21] := 155.4473;
   DATA[886,22] := 1.716721;
   DATA[886,23] := 948.5645;
   DATA[886,24] := 2.0;
   DATA[886,25] := 2.0;
   DATA[886,26] := 7.878942;
   DATA[886,27] := 144.5783;
   DATA[886,28] := 263.0415;
   DATA[886,29] := 12.07383;
   DATA[886,30] := 1.726865;
   DATA[886,31] := 1.280389;
   DATA[886,32] := 0.7353967;
   DATA[886,33] := 0.3081062;
   DATA[886,34] := 2.0;
   DATA[886,35] := 250.6729;
   DATA[886,36] := 1.746067;
   DATA[886,37] := 189.5187;
   DATA[886,38] := 0.000128152;
   DATA[886,39] := 1.0;
   DATA[887,0] := 2.536271;
   DATA[887,1] := 603.4719;
   DATA[887,2] := 2.0;
   DATA[887,3] := 1.0;
   DATA[887,4] := 262.3686;
   DATA[887,5] := 8.464048;
   DATA[887,6] := 315.1243;
   DATA[887,8] := 1.0;
   DATA[887,9] := 1.0;
   DATA[887,10] := 1.0;
   DATA[887,11] := 2.010372;
   DATA[887,13] := 1011.079;
   DATA[887,14] := 1.0;
   DATA[887,15] := 1.0;
   DATA[887,16] := 1.0;
   DATA[887,17] := 1.0;
   DATA[887,18] := 1.0;
   DATA[887,19] := 1.0;
   DATA[887,20] := 148.808;
   DATA[887,21] := 155.4473;
   DATA[887,22] := 1.716721;
   DATA[887,23] := 947.7954;
   DATA[887,24] := 2.0;
   DATA[887,25] := 2.0;
   DATA[887,26] := 7.878942;
   DATA[887,27] := 144.5783;
   DATA[887,28] := 263.0415;
   DATA[887,29] := 12.07383;
   DATA[887,30] := 1.726865;
   DATA[887,31] := 1.279365;
   DATA[887,32] := 0.7353967;
   DATA[887,33] := 0.3084265;
   DATA[887,34] := 2.0;
   DATA[887,35] := 250.5928;
   DATA[887,36] := 1.746067;
   DATA[887,37] := 189.2464;
   DATA[887,38] := 0.000128152;
   DATA[887,39] := 1.0;
   DATA[888,0] := 2.544278;
   DATA[888,1] := 603.6682;
   DATA[888,2] := 2.0;
   DATA[888,3] := 1.0;
   DATA[888,4] := 262.3686;
   DATA[888,5] := 8.464048;
   DATA[888,6] := 315.1243;
   DATA[888,8] := 1.0;
   DATA[888,9] := 1.0;
   DATA[888,10] := 1.0;
   DATA[888,11] := 2.010372;
   DATA[888,13] := 1010.919;
   DATA[888,14] := 1.0;
   DATA[888,15] := 1.0;
   DATA[888,16] := 1.0;
   DATA[888,17] := 1.0;
   DATA[888,18] := 1.0;
   DATA[888,19] := 1.0;
   DATA[888,20] := 148.808;
   DATA[888,21] := 155.4217;
   DATA[888,22] := 1.716721;
   DATA[888,23] := 947.757;
   DATA[888,24] := 2.0;
   DATA[888,25] := 2.0;
   DATA[888,26] := 7.878942;
   DATA[888,27] := 144.5783;
   DATA[888,28] := 263.0415;
   DATA[888,29] := 12.07383;
   DATA[888,30] := 1.726865;
   DATA[888,31] := 1.271295;
   DATA[888,32] := 0.7353967;
   DATA[888,33] := 0.3084265;
   DATA[888,34] := 2.0;
   DATA[888,35] := 250.4967;
   DATA[888,36] := 1.746067;
   DATA[888,37] := 189.2464;
   DATA[888,38] := 0.000128152;
   DATA[888,39] := 1.0;
   DATA[889,0] := 2.544278;
   DATA[889,1] := 603.6682;
   DATA[889,2] := 2.0;
   DATA[889,3] := 1.0;
   DATA[889,4] := 262.3686;
   DATA[889,5] := 8.463728;
   DATA[889,6] := 315.1243;
   DATA[889,8] := 1.0;
   DATA[889,9] := 1.0;
   DATA[889,10] := 1.0;
   DATA[889,11] := 2.010372;
   DATA[889,13] := 1011.039;
   DATA[889,14] := 1.0;
   DATA[889,15] := 1.0;
   DATA[889,16] := 1.0;
   DATA[889,17] := 1.0;
   DATA[889,18] := 1.0;
   DATA[889,19] := 1.0;
   DATA[889,20] := 148.808;
   DATA[889,21] := 155.4217;
   DATA[889,22] := 1.714286;
   DATA[889,23] := 947.1033;
   DATA[889,24] := 2.0;
   DATA[889,25] := 2.0;
   DATA[889,26] := 7.878942;
   DATA[889,27] := 144.5783;
   DATA[889,28] := 263.0415;
   DATA[889,29] := 12.07383;
   DATA[889,30] := 1.726865;
   DATA[889,31] := 1.262457;
   DATA[889,32] := 0.7353967;
   DATA[889,33] := 0.3075297;
   DATA[889,34] := 2.0;
   DATA[889,35] := 250.4967;
   DATA[889,36] := 1.746067;
   DATA[889,37] := 189.2464;
   DATA[889,38] := 0.000128152;
   DATA[889,39] := 1.0;
   DATA[890,0] := 2.548121;
   DATA[890,1] := 604.0607;
   DATA[890,2] := 2.0;
   DATA[890,3] := 1.0;
   DATA[890,4] := 262.3686;
   DATA[890,5] := 8.463728;
   DATA[890,6] := 315.1243;
   DATA[890,8] := 1.0;
   DATA[890,9] := 1.0;
   DATA[890,10] := 1.0;
   DATA[890,11] := 2.010372;
   DATA[890,13] := 1010.879;
   DATA[890,14] := 1.0;
   DATA[890,15] := 1.0;
   DATA[890,16] := 1.0;
   DATA[890,17] := 1.0;
   DATA[890,18] := 1.0;
   DATA[890,19] := 1.0;
   DATA[890,20] := 148.808;
   DATA[890,21] := 155.4217;
   DATA[890,22] := 1.712876;
   DATA[890,23] := 946.8342;
   DATA[890,24] := 2.0;
   DATA[890,25] := 2.0;
   DATA[890,26] := 7.878942;
   DATA[890,27] := 144.5783;
   DATA[890,28] := 263.0415;
   DATA[890,29] := 12.07383;
   DATA[890,30] := 1.725711;
   DATA[890,31] := 1.261176;
   DATA[890,32] := 0.7353967;
   DATA[890,33] := 0.3075297;
   DATA[890,34] := 2.0;
   DATA[890,35] := 250.4967;
   DATA[890,36] := 1.746067;
   DATA[890,37] := 189.2464;
   DATA[890,38] := 0.000128152;
   DATA[890,39] := 1.0;
   DATA[891,0] := 2.548121;
   DATA[891,1] := 604.257;
   DATA[891,2] := 2.0;
   DATA[891,3] := 1.0;
   DATA[891,4] := 262.3686;
   DATA[891,5] := 8.462126;
   DATA[891,6] := 315.1243;
   DATA[891,8] := 1.0;
   DATA[891,9] := 1.0;
   DATA[891,10] := 1.0;
   DATA[891,11] := 2.010372;
   DATA[891,13] := 1011.159;
   DATA[891,14] := 1.0;
   DATA[891,15] := 1.0;
   DATA[891,16] := 1.0;
   DATA[891,17] := 1.0;
   DATA[891,18] := 1.0;
   DATA[891,19] := 1.0;
   DATA[891,20] := 148.808;
   DATA[891,21] := 155.4217;
   DATA[891,22] := 1.712748;
   DATA[891,23] := 946.142;
   DATA[891,24] := 2.0;
   DATA[891,25] := 2.0;
   DATA[891,26] := 7.878942;
   DATA[891,27] := 144.5783;
   DATA[891,28] := 263.0415;
   DATA[891,29] := 12.07383;
   DATA[891,30] := 1.725711;
   DATA[891,31] := 1.267837;
   DATA[891,32] := 0.7353967;
   DATA[891,33] := 0.3086186;
   DATA[891,34] := 2.0;
   DATA[891,35] := 250.4967;
   DATA[891,36] := 1.746067;
   DATA[891,37] := 189.2464;
   DATA[891,38] := 0.000128152;
   DATA[891,39] := 1.0;
   DATA[892,0] := 2.548121;
   DATA[892,1] := 604.3354;
   DATA[892,2] := 2.0;
   DATA[892,3] := 1.0;
   DATA[892,4] := 262.3686;
   DATA[892,5] := 8.462126;
   DATA[892,6] := 315.3038;
   DATA[892,8] := 1.0;
   DATA[892,9] := 1.0;
   DATA[892,10] := 1.0;
   DATA[892,11] := 2.010372;
   DATA[892,13] := 1010.879;
   DATA[892,14] := 1.0;
   DATA[892,15] := 1.0;
   DATA[892,16] := 1.0;
   DATA[892,17] := 1.0;
   DATA[892,18] := 1.0;
   DATA[892,19] := 1.0;
   DATA[892,20] := 148.808;
   DATA[892,21] := 155.4217;
   DATA[892,22] := 1.712748;
   DATA[892,23] := 946.2189;
   DATA[892,24] := 2.0;
   DATA[892,25] := 2.0;
   DATA[892,26] := 7.878942;
   DATA[892,27] := 144.5783;
   DATA[892,28] := 263.0415;
   DATA[892,29] := 12.07383;
   DATA[892,30] := 1.725711;
   DATA[892,31] := 1.280902;
   DATA[892,32] := 0.7353967;
   DATA[892,33] := 0.3086186;
   DATA[892,34] := 2.0;
   DATA[892,35] := 250.4967;
   DATA[892,36] := 1.681991;
   DATA[892,37] := 189.2464;
   DATA[892,38] := 0.000128152;
   DATA[892,39] := 1.0;
   DATA[893,0] := 2.548121;
   DATA[893,1] := 604.3354;
   DATA[893,2] := 2.0;
   DATA[893,3] := 1.0;
   DATA[893,4] := 262.3686;
   DATA[893,5] := 8.462126;
   DATA[893,6] := 315.3294;
   DATA[893,8] := 1.0;
   DATA[893,9] := 1.0;
   DATA[893,10] := 1.0;
   DATA[893,11] := 2.010372;
   DATA[893,13] := 1010.959;
   DATA[893,14] := 1.0;
   DATA[893,15] := 1.0;
   DATA[893,16] := 1.0;
   DATA[893,17] := 1.0;
   DATA[893,18] := 1.0;
   DATA[893,19] := 1.0;
   DATA[893,20] := 148.808;
   DATA[893,21] := 155.4217;
   DATA[893,22] := 1.714798;
   DATA[893,23] := 945.6806;
   DATA[893,24] := 2.0;
   DATA[893,25] := 2.0;
   DATA[893,26] := 7.878942;
   DATA[893,27] := 144.5783;
   DATA[893,28] := 263.0415;
   DATA[893,29] := 12.07383;
   DATA[893,30] := 1.72507;
   DATA[893,31] := 1.282311;
   DATA[893,32] := 0.7353967;
   DATA[893,33] := 0.3086186;
   DATA[893,34] := 2.0;
   DATA[893,35] := 250.4967;
   DATA[893,36] := 1.681991;
   DATA[893,37] := 189.2464;
   DATA[893,38] := 0.000128152;
   DATA[893,39] := 1.0;
   DATA[894,0] := 2.548121;
   DATA[894,1] := 604.8458;
   DATA[894,2] := 2.0;
   DATA[894,3] := 1.0;
   DATA[894,4] := 262.3686;
   DATA[894,5] := 8.462126;
   DATA[894,6] := 315.3294;
   DATA[894,8] := 1.0;
   DATA[894,9] := 1.0;
   DATA[894,10] := 1.0;
   DATA[894,11] := 2.010372;
   DATA[894,13] := 1010.879;
   DATA[894,14] := 1.0;
   DATA[894,15] := 1.0;
   DATA[894,16] := 1.0;
   DATA[894,17] := 1.0;
   DATA[894,18] := 1.0;
   DATA[894,19] := 1.0;
   DATA[894,20] := 148.808;
   DATA[894,21] := 155.4217;
   DATA[894,22] := 1.714798;
   DATA[894,23] := 945.2576;
   DATA[894,24] := 2.0;
   DATA[894,25] := 2.0;
   DATA[894,26] := 7.878942;
   DATA[894,27] := 144.4501;
   DATA[894,28] := 263.0415;
   DATA[894,29] := 12.07383;
   DATA[894,30] := 1.72507;
   DATA[894,31] := 1.282311;
   DATA[894,32] := 0.7353967;
   DATA[894,33] := 0.3086186;
   DATA[894,34] := 2.0;
   DATA[894,35] := 250.4967;
   DATA[894,36] := 1.681991;
   DATA[894,37] := 189.2464;
   DATA[894,38] := 0.000128152;
   DATA[894,39] := 1.0;
   DATA[895,0] := 2.548121;
   DATA[895,1] := 605.1205;
   DATA[895,2] := 2.0;
   DATA[895,3] := 1.0;
   DATA[895,4] := 262.3686;
   DATA[895,5] := 8.462126;
   DATA[895,6] := 315.3294;
   DATA[895,8] := 1.0;
   DATA[895,9] := 1.0;
   DATA[895,10] := 1.0;
   DATA[895,11] := 2.010372;
   DATA[895,13] := 1010.919;
   DATA[895,14] := 1.0;
   DATA[895,15] := 1.0;
   DATA[895,16] := 1.0;
   DATA[895,17] := 1.0;
   DATA[895,18] := 1.0;
   DATA[895,19] := 1.0;
   DATA[895,20] := 148.808;
   DATA[895,21] := 155.4217;
   DATA[895,22] := 1.714798;
   DATA[895,23] := 944.7962;
   DATA[895,24] := 2.0;
   DATA[895,25] := 2.0;
   DATA[895,26] := 7.878942;
   DATA[895,27] := 144.4501;
   DATA[895,28] := 263.0415;
   DATA[895,29] := 12.07383;
   DATA[895,30] := 1.72507;
   DATA[895,31] := 1.273345;
   DATA[895,32] := 0.7353967;
   DATA[895,33] := 0.3086186;
   DATA[895,34] := 2.0;
   DATA[895,35] := 250.4967;
   DATA[895,36] := 1.681991;
   DATA[895,37] := 189.2464;
   DATA[895,38] := 0.000128152;
   DATA[895,39] := 1.0;
   DATA[896,0] := 2.544278;
   DATA[896,1] := 605.6308;
   DATA[896,2] := 2.0;
   DATA[896,3] := 1.0;
   DATA[896,4] := 262.3686;
   DATA[896,5] := 8.462126;
   DATA[896,6] := 315.3294;
   DATA[896,8] := 1.0;
   DATA[896,9] := 1.0;
   DATA[896,10] := 1.0;
   DATA[896,11] := 2.010372;
   DATA[896,13] := 1010.959;
   DATA[896,14] := 1.0;
   DATA[896,15] := 1.0;
   DATA[896,16] := 1.0;
   DATA[896,17] := 1.0;
   DATA[896,18] := 1.0;
   DATA[896,19] := 1.0;
   DATA[896,20] := 148.808;
   DATA[896,21] := 155.4217;
   DATA[896,22] := 1.714798;
   DATA[896,23] := 943.9503;
   DATA[896,24] := 2.0;
   DATA[896,25] := 2.0;
   DATA[896,26] := 7.878942;
   DATA[896,27] := 144.4501;
   DATA[896,28] := 263.0415;
   DATA[896,29] := 12.07383;
   DATA[896,30] := 1.726096;
   DATA[896,31] := 1.271935;
   DATA[896,32] := 0.7353967;
   DATA[896,33] := 0.3086186;
   DATA[896,34] := 2.0;
   DATA[896,35] := 250.4967;
   DATA[896,36] := 1.681991;
   DATA[896,37] := 189.2464;
   DATA[896,38] := 0.000128152;
   DATA[896,39] := 1.0;
   DATA[897,0] := 2.544278;
   DATA[897,1] := 606.0626;
   DATA[897,2] := 2.0;
   DATA[897,3] := 1.0;
   DATA[897,4] := 262.3686;
   DATA[897,5] := 8.462126;
   DATA[897,6] := 315.3294;
   DATA[897,8] := 1.0;
   DATA[897,9] := 1.0;
   DATA[897,10] := 1.0;
   DATA[897,11] := 2.010372;
   DATA[897,13] := 1011.039;
   DATA[897,14] := 1.0;
   DATA[897,15] := 1.0;
   DATA[897,16] := 1.0;
   DATA[897,17] := 1.0;
   DATA[897,18] := 1.0;
   DATA[897,19] := 1.0;
   DATA[897,20] := 148.808;
   DATA[897,21] := 155.4217;
   DATA[897,22] := 1.714798;
   DATA[897,23] := 943.4888;
   DATA[897,24] := 2.0;
   DATA[897,25] := 2.0;
   DATA[897,26] := 7.878942;
   DATA[897,27] := 144.4501;
   DATA[897,28] := 263.0415;
   DATA[897,29] := 12.07383;
   DATA[897,30] := 1.726609;
   DATA[897,31] := 1.277443;
   DATA[897,32] := 0.7353967;
   DATA[897,33] := 0.3086186;
   DATA[897,34] := 2.0;
   DATA[897,35] := 250.4967;
   DATA[897,36] := 1.681991;
   DATA[897,37] := 189.2464;
   DATA[897,38] := 0.000128152;
   DATA[897,39] := 1.0;
   DATA[898,0] := 2.544278;
   DATA[898,1] := 606.0626;
   DATA[898,2] := 2.0;
   DATA[898,3] := 1.0;
   DATA[898,4] := 262.3686;
   DATA[898,5] := 8.461164;
   DATA[898,6] := 315.3294;
   DATA[898,8] := 1.0;
   DATA[898,9] := 1.0;
   DATA[898,10] := 1.0;
   DATA[898,11] := 2.010372;
   DATA[898,13] := 1011.039;
   DATA[898,14] := 1.0;
   DATA[898,15] := 1.0;
   DATA[898,16] := 1.0;
   DATA[898,17] := 1.0;
   DATA[898,18] := 1.0;
   DATA[898,19] := 1.0;
   DATA[898,20] := 148.808;
   DATA[898,21] := 155.4217;
   DATA[898,22] := 1.714798;
   DATA[898,23] := 943.1043;
   DATA[898,24] := 2.0;
   DATA[898,25] := 2.0;
   DATA[898,26] := 7.878942;
   DATA[898,27] := 144.4501;
   DATA[898,28] := 263.0415;
   DATA[898,29] := 12.07383;
   DATA[898,30] := 1.726609;
   DATA[898,31] := 1.276162;
   DATA[898,32] := 0.7353967;
   DATA[898,33] := 0.3086186;
   DATA[898,34] := 2.0;
   DATA[898,35] := 250.4967;
   DATA[898,36] := 1.681991;
   DATA[898,37] := 189.2464;
   DATA[898,38] := 0.000128152;
   DATA[898,39] := 1.0;
   DATA[899,0] := 2.551645;
   DATA[899,1] := 606.2589;
   DATA[899,2] := 2.0;
   DATA[899,3] := 1.0;
   DATA[899,4] := 262.3686;
   DATA[899,5] := 8.459562;
   DATA[899,6] := 315.3294;
   DATA[899,8] := 1.0;
   DATA[899,9] := 1.0;
   DATA[899,10] := 1.0;
   DATA[899,11] := 2.010372;
   DATA[899,13] := 1010.718;
   DATA[899,14] := 1.0;
   DATA[899,15] := 1.0;
   DATA[899,16] := 1.0;
   DATA[899,17] := 1.0;
   DATA[899,18] := 1.0;
   DATA[899,19] := 1.0;
   DATA[899,20] := 148.808;
   DATA[899,21] := 155.4217;
   DATA[899,22] := 1.714798;
   DATA[899,23] := 942.989;
   DATA[899,24] := 2.0;
   DATA[899,25] := 2.0;
   DATA[899,26] := 7.878942;
   DATA[899,27] := 144.4501;
   DATA[899,28] := 263.0415;
   DATA[899,29] := 12.07383;
   DATA[899,30] := 1.726609;
   DATA[899,31] := 1.282567;
   DATA[899,32] := 0.7353967;
   DATA[899,33] := 0.3084265;
   DATA[899,34] := 2.0;
   DATA[899,35] := 250.4326;
   DATA[899,36] := 1.681991;
   DATA[899,37] := 189.2464;
   DATA[899,38] := 0.000128152;
   DATA[899,39] := 1.0;
   DATA[900,0] := 2.551645;
   DATA[900,1] := 606.4158;
   DATA[900,2] := 2.0;
   DATA[900,3] := 1.0;
   DATA[900,4] := 262.3686;
   DATA[900,5] := 8.459562;
   DATA[900,6] := 315.3294;
   DATA[900,8] := 1.0;
   DATA[900,9] := 1.0;
   DATA[900,10] := 1.0;
   DATA[900,11] := 2.010372;
   DATA[900,13] := 1010.518;
   DATA[900,14] := 1.0;
   DATA[900,15] := 1.0;
   DATA[900,16] := 1.0;
   DATA[900,17] := 1.0;
   DATA[900,18] := 1.0;
   DATA[900,19] := 1.0;
   DATA[900,20] := 148.808;
   DATA[900,21] := 155.4217;
   DATA[900,22] := 1.713517;
   DATA[900,23] := 942.6429;
   DATA[900,24] := 2.0;
   DATA[900,25] := 2.0;
   DATA[900,26] := 7.878942;
   DATA[900,27] := 144.4501;
   DATA[900,28] := 263.0415;
   DATA[900,29] := 12.07383;
   DATA[900,30] := 1.726993;
   DATA[900,31] := 1.301012;
   DATA[900,32] := 0.7353967;
   DATA[900,33] := 0.3084265;
   DATA[900,34] := 2.0;
   DATA[900,35] := 250.4326;
   DATA[900,36] := 1.681991;
   DATA[900,37] := 189.2464;
   DATA[900,38] := 0.000128152;
   DATA[900,39] := 1.0;
   DATA[901,0] := 2.551645;
   DATA[901,1] := 606.4551;
   DATA[901,2] := 2.0;
   DATA[901,3] := 1.0;
   DATA[901,4] := 262.3686;
   DATA[901,5] := 8.459562;
   DATA[901,6] := 315.3294;
   DATA[901,8] := 1.0;
   DATA[901,9] := 1.0;
   DATA[901,10] := 1.0;
   DATA[901,11] := 2.010372;
   DATA[901,13] := 1011.119;
   DATA[901,14] := 1.0;
   DATA[901,15] := 1.0;
   DATA[901,16] := 1.0;
   DATA[901,17] := 1.0;
   DATA[901,18] := 1.0;
   DATA[901,19] := 1.0;
   DATA[901,20] := 148.808;
   DATA[901,21] := 155.4217;
   DATA[901,22] := 1.713004;
   DATA[901,23] := 942.1815;
   DATA[901,24] := 2.0;
   DATA[901,25] := 2.0;
   DATA[901,26] := 7.878942;
   DATA[901,27] := 144.4501;
   DATA[901,28] := 263.0415;
   DATA[901,29] := 12.07383;
   DATA[901,30] := 1.726993;
   DATA[901,31] := 1.302293;
   DATA[901,32] := 0.7353967;
   DATA[901,33] := 0.3084265;
   DATA[901,34] := 2.0;
   DATA[901,35] := 250.4326;
   DATA[901,36] := 1.681991;
   DATA[901,37] := 189.2464;
   DATA[901,38] := 0.000128152;
   DATA[901,39] := 1.0;
   DATA[902,0] := 2.555168;
   DATA[902,1] := 606.4944;
   DATA[902,2] := 2.0;
   DATA[902,3] := 1.0;
   DATA[902,4] := 262.3686;
   DATA[902,5] := 8.459562;
   DATA[902,6] := 315.3294;
   DATA[902,8] := 1.0;
   DATA[902,9] := 1.0;
   DATA[902,10] := 1.0;
   DATA[902,11] := 2.010372;
   DATA[902,13] := 1011.079;
   DATA[902,14] := 1.0;
   DATA[902,15] := 1.0;
   DATA[902,16] := 1.0;
   DATA[902,17] := 1.0;
   DATA[902,18] := 1.0;
   DATA[902,19] := 1.0;
   DATA[902,20] := 148.808;
   DATA[902,21] := 155.4217;
   DATA[902,22] := 1.713004;
   DATA[902,23] := 941.8354;
   DATA[902,24] := 2.0;
   DATA[902,25] := 2.0;
   DATA[902,26] := 7.878942;
   DATA[902,27] := 144.2707;
   DATA[902,28] := 263.0415;
   DATA[902,29] := 12.07383;
   DATA[902,30] := 1.726993;
   DATA[902,31] := 1.302293;
   DATA[902,32] := 0.7353967;
   DATA[902,33] := 0.3084265;
   DATA[902,34] := 2.0;
   DATA[902,35] := 250.4326;
   DATA[902,36] := 1.681991;
   DATA[902,37] := 189.2464;
   DATA[902,38] := 0.000128152;
   DATA[902,39] := 1.0;
   DATA[903,0] := 2.555168;
   DATA[903,1] := 606.9261;
   DATA[903,2] := 2.0;
   DATA[903,3] := 1.0;
   DATA[903,4] := 262.5288;
   DATA[903,5] := 8.459562;
   DATA[903,6] := 315.3294;
   DATA[903,8] := 1.0;
   DATA[903,9] := 1.0;
   DATA[903,10] := 1.0;
   DATA[903,11] := 2.010372;
   DATA[903,13] := 1011.159;
   DATA[903,14] := 1.0;
   DATA[903,15] := 1.0;
   DATA[903,16] := 1.0;
   DATA[903,17] := 1.0;
   DATA[903,18] := 1.0;
   DATA[903,19] := 1.0;
   DATA[903,20] := 148.808;
   DATA[903,21] := 155.4217;
   DATA[903,22] := 1.711595;
   DATA[903,23] := 941.1049;
   DATA[903,24] := 2.0;
   DATA[903,25] := 2.0;
   DATA[903,26] := 7.878942;
   DATA[903,27] := 144.2707;
   DATA[903,28] := 263.0415;
   DATA[903,29] := 12.07383;
   DATA[903,30] := 1.724814;
   DATA[903,31] := 1.296273;
   DATA[903,32] := 0.7353967;
   DATA[903,33] := 0.3084265;
   DATA[903,34] := 2.0;
   DATA[903,35] := 250.4326;
   DATA[903,36] := 1.681991;
   DATA[903,37] := 189.2464;
   DATA[903,38] := 0.000128152;
   DATA[903,39] := 1.0;
   DATA[904,0] := 2.555168;
   DATA[904,1] := 607.829;
   DATA[904,2] := 2.0;
   DATA[904,3] := 1.0;
   DATA[904,4] := 262.5288;
   DATA[904,5] := 8.459562;
   DATA[904,6] := 315.3294;
   DATA[904,8] := 1.0;
   DATA[904,9] := 1.0;
   DATA[904,10] := 1.0;
   DATA[904,11] := 2.010372;
   DATA[904,13] := 1011.039;
   DATA[904,14] := 1.0;
   DATA[904,15] := 1.0;
   DATA[904,16] := 1.0;
   DATA[904,17] := 1.0;
   DATA[904,18] := 1.0;
   DATA[904,19] := 1.0;
   DATA[904,20] := 148.808;
   DATA[904,21] := 155.4217;
   DATA[904,22] := 1.714029;
   DATA[904,23] := 940.6819;
   DATA[904,24] := 2.0;
   DATA[904,25] := 2.0;
   DATA[904,26] := 7.878942;
   DATA[904,27] := 144.2707;
   DATA[904,28] := 263.0415;
   DATA[904,29] := 12.07383;
   DATA[904,30] := 1.724814;
   DATA[904,31] := 1.299859;
   DATA[904,32] := 0.7353967;
   DATA[904,33] := 0.3084265;
   DATA[904,34] := 2.0;
   DATA[904,35] := 250.4326;
   DATA[904,36] := 1.681991;
   DATA[904,37] := 189.2464;
   DATA[904,38] := 0.000128152;
   DATA[904,39] := 1.0;
   DATA[905,0] := 2.555168;
   DATA[905,1] := 608.2607;
   DATA[905,2] := 2.0;
   DATA[905,3] := 1.0;
   DATA[905,4] := 262.5288;
   DATA[905,5] := 8.459562;
   DATA[905,6] := 315.3294;
   DATA[905,8] := 1.0;
   DATA[905,9] := 1.0;
   DATA[905,10] := 1.0;
   DATA[905,11] := 2.010372;
   DATA[905,13] := 1010.839;
   DATA[905,14] := 1.0;
   DATA[905,15] := 1.0;
   DATA[905,16] := 1.0;
   DATA[905,17] := 1.0;
   DATA[905,18] := 1.0;
   DATA[905,19] := 1.0;
   DATA[905,20] := 148.808;
   DATA[905,21] := 155.4217;
   DATA[905,22] := 1.714158;
   DATA[905,23] := 939.9513;
   DATA[905,24] := 2.0;
   DATA[905,25] := 2.0;
   DATA[905,26] := 7.878942;
   DATA[905,27] := 144.2707;
   DATA[905,28] := 263.0415;
   DATA[905,29] := 12.07383;
   DATA[905,30] := 1.724814;
   DATA[905,31] := 1.305239;
   DATA[905,32] := 0.7353967;
   DATA[905,33] := 0.3084265;
   DATA[905,34] := 2.0;
   DATA[905,35] := 250.4326;
   DATA[905,36] := 1.681991;
   DATA[905,37] := 189.2464;
   DATA[905,38] := 0.000128152;
   DATA[905,39] := 1.0;
   DATA[906,0] := 2.550364;
   DATA[906,1] := 609.0458;
   DATA[906,2] := 2.0;
   DATA[906,3] := 1.0;
   DATA[906,4] := 262.5288;
   DATA[906,5] := 8.459562;
   DATA[906,6] := 315.3294;
   DATA[906,8] := 1.0;
   DATA[906,9] := 1.0;
   DATA[906,10] := 1.0;
   DATA[906,11] := 2.010372;
   DATA[906,13] := 1010.959;
   DATA[906,14] := 1.0;
   DATA[906,15] := 1.0;
   DATA[906,16] := 1.0;
   DATA[906,17] := 1.0;
   DATA[906,18] := 1.0;
   DATA[906,19] := 1.0;
   DATA[906,20] := 148.808;
   DATA[906,21] := 155.4217;
   DATA[906,22] := 1.714158;
   DATA[906,23] := 939.4514;
   DATA[906,24] := 2.0;
   DATA[906,25] := 2.0;
   DATA[906,26] := 7.878942;
   DATA[906,27] := 144.2707;
   DATA[906,28] := 263.0415;
   DATA[906,29] := 12.07383;
   DATA[906,30] := 1.726737;
   DATA[906,31] := 1.311643;
   DATA[906,32] := 0.7353967;
   DATA[906,33] := 0.3084265;
   DATA[906,34] := 2.0;
   DATA[906,35] := 250.4326;
   DATA[906,36] := 1.681991;
   DATA[906,37] := 189.2464;
   DATA[906,38] := 0.000128152;
   DATA[906,39] := 1.0;
   DATA[907,0] := 2.550364;
   DATA[907,1] := 609.8701;
   DATA[907,2] := 2.0;
   DATA[907,3] := 1.0;
   DATA[907,4] := 262.5288;
   DATA[907,5] := 8.459562;
   DATA[907,6] := 315.3294;
   DATA[907,8] := 1.0;
   DATA[907,9] := 1.0;
   DATA[907,10] := 1.0;
   DATA[907,11] := 2.010372;
   DATA[907,13] := 1011.119;
   DATA[907,14] := 1.0;
   DATA[907,15] := 1.0;
   DATA[907,16] := 1.0;
   DATA[907,17] := 1.0;
   DATA[907,18] := 1.0;
   DATA[907,19] := 1.0;
   DATA[907,20] := 148.808;
   DATA[907,21] := 155.4217;
   DATA[907,22] := 1.714158;
   DATA[907,23] := 939.4514;
   DATA[907,24] := 2.0;
   DATA[907,25] := 2.0;
   DATA[907,26] := 7.878942;
   DATA[907,27] := 144.2707;
   DATA[907,28] := 263.0415;
   DATA[907,29] := 12.07383;
   DATA[907,30] := 1.726737;
   DATA[907,31] := 1.31254;
   DATA[907,32] := 0.7353967;
   DATA[907,33] := 0.3084265;
   DATA[907,34] := 2.0;
   DATA[907,35] := 250.4326;
   DATA[907,36] := 1.681991;
   DATA[907,37] := 189.2464;
   DATA[907,38] := 0.000128152;
   DATA[907,39] := 1.0;
   DATA[908,0] := 2.550364;
   DATA[908,1] := 610.5767;
   DATA[908,2] := 2.0;
   DATA[908,3] := 1.0;
   DATA[908,4] := 262.5288;
   DATA[908,5] := 8.459562;
   DATA[908,6] := 315.3294;
   DATA[908,8] := 1.0;
   DATA[908,9] := 1.0;
   DATA[908,10] := 1.0;
   DATA[908,11] := 2.010372;
   DATA[908,13] := 1011.079;
   DATA[908,14] := 1.0;
   DATA[908,15] := 1.0;
   DATA[908,16] := 1.0;
   DATA[908,17] := 1.0;
   DATA[908,18] := 1.0;
   DATA[908,19] := 1.0;
   DATA[908,20] := 148.808;
   DATA[908,21] := 155.4217;
   DATA[908,22] := 1.714158;
   DATA[908,23] := 939.3745;
   DATA[908,24] := 2.0;
   DATA[908,25] := 2.0;
   DATA[908,26] := 7.878942;
   DATA[908,27] := 144.2707;
   DATA[908,28] := 263.0415;
   DATA[908,29] := 12.07383;
   DATA[908,30] := 1.726737;
   DATA[908,31] := 1.303318;
   DATA[908,32] := 0.7353967;
   DATA[908,33] := 0.3084265;
   DATA[908,34] := 2.0;
   DATA[908,35] := 250.4326;
   DATA[908,36] := 1.681991;
   DATA[908,37] := 189.2464;
   DATA[908,38] := 0.000128152;
   DATA[908,39] := 1.0;
   DATA[909,0] := 2.550364;
   DATA[909,1] := 611.1262;
   DATA[909,2] := 2.0;
   DATA[909,3] := 1.0;
   DATA[909,4] := 262.5288;
   DATA[909,5] := 8.459562;
   DATA[909,6] := 315.3294;
   DATA[909,8] := 1.0;
   DATA[909,9] := 1.0;
   DATA[909,10] := 1.0;
   DATA[909,11] := 2.010372;
   DATA[909,13] := 1011.279;
   DATA[909,14] := 1.0;
   DATA[909,15] := 1.0;
   DATA[909,16] := 1.0;
   DATA[909,17] := 1.0;
   DATA[909,18] := 1.0;
   DATA[909,19] := 1.0;
   DATA[909,20] := 148.808;
   DATA[909,21] := 155.4217;
   DATA[909,22] := 1.712748;
   DATA[909,23] := 939.2592;
   DATA[909,24] := 2.0;
   DATA[909,25] := 2.0;
   DATA[909,26] := 7.878942;
   DATA[909,27] := 144.2707;
   DATA[909,28] := 263.0415;
   DATA[909,29] := 12.07383;
   DATA[909,30] := 1.726737;
   DATA[909,31] := 1.301652;
   DATA[909,32] := 0.7353967;
   DATA[909,33] := 0.3084265;
   DATA[909,34] := 2.0;
   DATA[909,35] := 250.4326;
   DATA[909,36] := 1.681991;
   DATA[909,37] := 189.2464;
   DATA[909,38] := 0.000128152;
   DATA[909,39] := 1.0;
   DATA[910,0] := 2.551645;
   DATA[910,1] := 611.9897;
   DATA[910,2] := 2.0;
   DATA[910,3] := 1.0;
   DATA[910,4] := 262.5288;
   DATA[910,5] := 8.459562;
   DATA[910,6] := 315.3294;
   DATA[910,8] := 1.0;
   DATA[910,9] := 1.0;
   DATA[910,10] := 1.0;
   DATA[910,11] := 2.010372;
   DATA[910,13] := 1011.279;
   DATA[910,14] := 1.0;
   DATA[910,15] := 1.0;
   DATA[910,16] := 1.0;
   DATA[910,17] := 1.0;
   DATA[910,18] := 1.0;
   DATA[910,19] := 1.0;
   DATA[910,20] := 148.808;
   DATA[910,21] := 155.4217;
   DATA[910,22] := 1.711466;
   DATA[910,23] := 938.7208;
   DATA[910,24] := 2.0;
   DATA[910,25] := 2.0;
   DATA[910,26] := 7.878942;
   DATA[910,27] := 144.2707;
   DATA[910,28] := 263.0415;
   DATA[910,29] := 12.07383;
   DATA[910,30] := 1.726737;
   DATA[910,31] := 1.306904;
   DATA[910,32] := 0.7353967;
   DATA[910,33] := 0.3084265;
   DATA[910,34] := 2.0;
   DATA[910,35] := 250.4326;
   DATA[910,36] := 1.681991;
   DATA[910,37] := 189.2464;
   DATA[910,38] := 0.000128152;
   DATA[910,39] := 1.0;
   DATA[911,0] := 2.551645;
   DATA[911,1] := 611.9897;
   DATA[911,2] := 2.0;
   DATA[911,3] := 1.0;
   DATA[911,4] := 262.5288;
   DATA[911,5] := 8.459562;
   DATA[911,6] := 315.3294;
   DATA[911,8] := 1.0;
   DATA[911,9] := 1.0;
   DATA[911,10] := 1.0;
   DATA[911,11] := 2.010372;
   DATA[911,13] := 1011.279;
   DATA[911,14] := 1.0;
   DATA[911,15] := 1.0;
   DATA[911,16] := 1.0;
   DATA[911,17] := 1.0;
   DATA[911,18] := 1.0;
   DATA[911,19] := 1.0;
   DATA[911,20] := 148.808;
   DATA[911,21] := 155.4217;
   DATA[911,22] := 1.711466;
   DATA[911,23] := 938.7208;
   DATA[911,24] := 2.0;
   DATA[911,25] := 2.0;
   DATA[911,26] := 7.878942;
   DATA[911,27] := 144.2707;
   DATA[911,28] := 263.0415;
   DATA[911,29] := 12.07383;
   DATA[911,30] := 1.726737;
   DATA[911,31] := 1.306904;
   DATA[911,32] := 0.7353967;
   DATA[911,33] := 0.3084265;
   DATA[911,34] := 2.0;
   DATA[911,35] := 250.4326;
   DATA[911,36] := 1.681991;
   DATA[911,37] := 189.2464;
   DATA[911,38] := 0.000128152;
   DATA[911,39] := 1.0;
   DATA[912,0] := 2.554847;
   DATA[912,1] := 612.7748;
   DATA[912,2] := 2.0;
   DATA[912,3] := 1.0;
   DATA[912,4] := 262.5288;
   DATA[912,5] := 8.459562;
   DATA[912,6] := 315.3294;
   DATA[912,8] := 1.0;
   DATA[912,9] := 1.0;
   DATA[912,10] := 1.0;
   DATA[912,11] := 2.010372;
   DATA[912,13] := 1010.959;
   DATA[912,14] := 1.0;
   DATA[912,15] := 1.0;
   DATA[912,16] := 1.0;
   DATA[912,17] := 1.0;
   DATA[912,18] := 1.0;
   DATA[912,19] := 1.0;
   DATA[912,20] := 148.808;
   DATA[912,21] := 155.4217;
   DATA[912,22] := 1.711466;
   DATA[912,23] := 938.3363;
   DATA[912,24] := 2.0;
   DATA[912,25] := 2.0;
   DATA[912,26] := 7.878942;
   DATA[912,27] := 144.2707;
   DATA[912,28] := 263.0415;
   DATA[912,29] := 12.07383;
   DATA[912,30] := 1.726737;
   DATA[912,31] := 1.303702;
   DATA[912,32] := 0.7353967;
   DATA[912,33] := 0.3084265;
   DATA[912,34] := 2.0;
   DATA[912,35] := 250.4166;
   DATA[912,36] := 1.681991;
   DATA[912,37] := 189.2464;
   DATA[912,38] := 0.000128152;
   DATA[912,39] := 1.0;
   DATA[913,0] := 2.554847;
   DATA[913,1] := 613.2851;
   DATA[913,2] := 2.0;
   DATA[913,3] := 1.0;
   DATA[913,4] := 262.5288;
   DATA[913,5] := 8.459562;
   DATA[913,6] := 315.3294;
   DATA[913,8] := 1.0;
   DATA[913,9] := 1.0;
   DATA[913,10] := 1.0;
   DATA[913,11] := 2.010372;
   DATA[913,13] := 1010.879;
   DATA[913,14] := 1.0;
   DATA[913,15] := 1.0;
   DATA[913,16] := 1.0;
   DATA[913,17] := 1.0;
   DATA[913,18] := 1.0;
   DATA[913,19] := 1.0;
   DATA[913,20] := 148.808;
   DATA[913,21] := 155.4217;
   DATA[913,22] := 1.711466;
   DATA[913,23] := 938.3363;
   DATA[913,24] := 2.0;
   DATA[913,25] := 2.0;
   DATA[913,26] := 7.878942;
   DATA[913,27] := 144.2707;
   DATA[913,28] := 263.0415;
   DATA[913,29] := 12.07383;
   DATA[913,30] := 1.726737;
   DATA[913,31] := 1.301524;
   DATA[913,32] := 0.7353967;
   DATA[913,33] := 0.3084265;
   DATA[913,34] := 2.0;
   DATA[913,35] := 250.4166;
   DATA[913,36] := 1.681991;
   DATA[913,37] := 189.2464;
   DATA[913,38] := 0.000128152;
   DATA[913,39] := 1.0;
   DATA[914,0] := 2.554847;
   DATA[914,1] := 613.9916;
   DATA[914,2] := 2.0;
   DATA[914,3] := 1.0;
   DATA[914,4] := 262.5288;
   DATA[914,5] := 8.459562;
   DATA[914,6] := 315.3294;
   DATA[914,8] := 1.0;
   DATA[914,9] := 1.0;
   DATA[914,10] := 1.0;
   DATA[914,11] := 2.010372;
   DATA[914,13] := 1010.638;
   DATA[914,14] := 1.0;
   DATA[914,15] := 1.0;
   DATA[914,16] := 1.0;
   DATA[914,17] := 1.0;
   DATA[914,18] := 1.0;
   DATA[914,19] := 1.0;
   DATA[914,20] := 148.808;
   DATA[914,21] := 155.4217;
   DATA[914,22] := 1.711466;
   DATA[914,23] := 937.7595;
   DATA[914,24] := 2.0;
   DATA[914,25] := 2.0;
   DATA[914,26] := 7.878942;
   DATA[914,27] := 144.2707;
   DATA[914,28] := 263.0415;
   DATA[914,29] := 12.07383;
   DATA[914,30] := 1.726737;
   DATA[914,31] := 1.297297;
   DATA[914,32] := 0.7353967;
   DATA[914,33] := 0.3084265;
   DATA[914,34] := 2.0;
   DATA[914,35] := 250.4166;
   DATA[914,36] := 1.681991;
   DATA[914,37] := 189.2464;
   DATA[914,38] := 0.000128152;
   DATA[914,39] := 1.0;
   DATA[915,0] := 2.554847;
   DATA[915,1] := 614.5804;
   DATA[915,2] := 2.0;
   DATA[915,3] := 1.0;
   DATA[915,4] := 262.5288;
   DATA[915,5] := 8.459562;
   DATA[915,6] := 315.3294;
   DATA[915,8] := 1.0;
   DATA[915,9] := 1.0;
   DATA[915,10] := 1.0;
   DATA[915,11] := 2.010372;
   DATA[915,13] := 1010.718;
   DATA[915,14] := 1.0;
   DATA[915,15] := 1.0;
   DATA[915,16] := 1.0;
   DATA[915,17] := 1.0;
   DATA[915,18] := 1.0;
   DATA[915,19] := 1.0;
   DATA[915,20] := 148.808;
   DATA[915,21] := 155.4217;
   DATA[915,22] := 1.711595;
   DATA[915,23] := 937.3366;
   DATA[915,24] := 2.0;
   DATA[915,25] := 2.0;
   DATA[915,26] := 7.878942;
   DATA[915,27] := 144.322;
   DATA[915,28] := 263.0415;
   DATA[915,29] := 12.07383;
   DATA[915,30] := 1.726096;
   DATA[915,31] := 1.287562;
   DATA[915,32] := 0.7353967;
   DATA[915,33] := 0.3084265;
   DATA[915,34] := 2.0;
   DATA[915,35] := 250.4166;
   DATA[915,36] := 1.681991;
   DATA[915,37] := 189.2464;
   DATA[915,38] := 0.000128152;
   DATA[915,39] := 1.0;
   DATA[916,0] := 2.54652;
   DATA[916,1] := 615.1693;
   DATA[916,2] := 2.0;
   DATA[916,3] := 1.0;
   DATA[916,4] := 262.5288;
   DATA[916,5] := 8.459562;
   DATA[916,6] := 315.3294;
   DATA[916,8] := 1.0;
   DATA[916,9] := 1.0;
   DATA[916,10] := 1.0;
   DATA[916,11] := 2.010372;
   DATA[916,13] := 1010.718;
   DATA[916,14] := 1.0;
   DATA[916,15] := 1.0;
   DATA[916,16] := 1.0;
   DATA[916,17] := 1.0;
   DATA[916,18] := 1.0;
   DATA[916,19] := 1.0;
   DATA[916,20] := 148.808;
   DATA[916,21] := 155.4217;
   DATA[916,22] := 1.712235;
   DATA[916,23] := 936.7598;
   DATA[916,24] := 2.0;
   DATA[916,25] := 2.0;
   DATA[916,26] := 7.878942;
   DATA[916,27] := 144.322;
   DATA[916,28] := 263.0415;
   DATA[916,29] := 12.07383;
   DATA[916,30] := 1.72443;
   DATA[916,31] := 1.291789;
   DATA[916,32] := 0.7353967;
   DATA[916,33] := 0.3084265;
   DATA[916,34] := 2.0;
   DATA[916,35] := 250.4166;
   DATA[916,36] := 1.681991;
   DATA[916,37] := 189.2464;
   DATA[916,38] := 0.000128152;
   DATA[916,39] := 1.0;
   DATA[917,0] := 2.540115;
   DATA[917,1] := 615.8365;
   DATA[917,2] := 2.0;
   DATA[917,3] := 1.0;
   DATA[917,4] := 262.5288;
   DATA[917,5] := 8.459562;
   DATA[917,6] := 315.3294;
   DATA[917,8] := 1.0;
   DATA[917,9] := 1.0;
   DATA[917,10] := 1.0;
   DATA[917,11] := 2.010372;
   DATA[917,13] := 1011.119;
   DATA[917,14] := 1.0;
   DATA[917,15] := 1.0;
   DATA[917,16] := 1.0;
   DATA[917,17] := 1.0;
   DATA[917,18] := 1.0;
   DATA[917,19] := 1.0;
   DATA[917,20] := 148.808;
   DATA[917,21] := 155.4217;
   DATA[917,22] := 1.71608;
   DATA[917,23] := 936.4522;
   DATA[917,24] := 2.0;
   DATA[917,25] := 2.0;
   DATA[917,26] := 7.878942;
   DATA[917,27] := 144.322;
   DATA[917,28] := 263.0415;
   DATA[917,29] := 12.07383;
   DATA[917,30] := 1.72443;
   DATA[917,31] := 1.291789;
   DATA[917,32] := 0.7353967;
   DATA[917,33] := 0.3084265;
   DATA[917,34] := 2.0;
   DATA[917,35] := 250.4166;
   DATA[917,36] := 1.681991;
   DATA[917,37] := 189.2464;
   DATA[917,38] := 0.000128152;
   DATA[917,39] := 1.0;
   DATA[918,0] := 2.538513;
   DATA[918,1] := 616.0328;
   DATA[918,2] := 2.0;
   DATA[918,3] := 1.0;
   DATA[918,4] := 262.5288;
   DATA[918,5] := 8.459562;
   DATA[918,6] := 315.3294;
   DATA[918,8] := 1.0;
   DATA[918,9] := 1.0;
   DATA[918,10] := 1.0;
   DATA[918,11] := 2.010372;
   DATA[918,13] := 1011.039;
   DATA[918,14] := 1.0;
   DATA[918,15] := 1.0;
   DATA[918,16] := 1.0;
   DATA[918,17] := 1.0;
   DATA[918,18] := 1.0;
   DATA[918,19] := 1.0;
   DATA[918,20] := 148.808;
   DATA[918,21] := 155.4217;
   DATA[918,22] := 1.716592;
   DATA[918,23] := 936.2599;
   DATA[918,24] := 2.0;
   DATA[918,25] := 2.0;
   DATA[918,26] := 7.878942;
   DATA[918,27] := 144.527;
   DATA[918,28] := 263.0415;
   DATA[918,29] := 12.07383;
   DATA[918,30] := 1.72443;
   DATA[918,31] := 1.282567;
   DATA[918,32] := 0.7353967;
   DATA[918,33] := 0.3084265;
   DATA[918,34] := 2.0;
   DATA[918,35] := 250.3204;
   DATA[918,36] := 1.681991;
   DATA[918,37] := 189.2464;
   DATA[918,38] := 0.000128152;
   DATA[918,39] := 1.0;
   DATA[919,0] := 2.538513;
   DATA[919,1] := 616.3468;
   DATA[919,2] := 2.0;
   DATA[919,3] := 1.0;
   DATA[919,4] := 262.5288;
   DATA[919,5] := 8.459562;
   DATA[919,6] := 315.4576;
   DATA[919,8] := 1.0;
   DATA[919,9] := 1.0;
   DATA[919,10] := 1.0;
   DATA[919,11] := 2.010372;
   DATA[919,13] := 1011.119;
   DATA[919,14] := 1.0;
   DATA[919,15] := 1.0;
   DATA[919,16] := 1.0;
   DATA[919,17] := 1.0;
   DATA[919,18] := 1.0;
   DATA[919,19] := 1.0;
   DATA[919,20] := 148.808;
   DATA[919,21] := 155.4217;
   DATA[919,22] := 1.717489;
   DATA[919,23] := 935.9908;
   DATA[919,24] := 2.0;
   DATA[919,25] := 2.0;
   DATA[919,26] := 7.878942;
   DATA[919,27] := 144.527;
   DATA[919,28] := 263.0415;
   DATA[919,29] := 12.07383;
   DATA[919,30] := 1.72443;
   DATA[919,31] := 1.281927;
   DATA[919,32] := 0.7353967;
   DATA[919,33] := 0.3084265;
   DATA[919,34] := 2.0;
   DATA[919,35] := 250.3204;
   DATA[919,36] := 1.681991;
   DATA[919,37] := 189.2464;
   DATA[919,38] := 0.000128152;
   DATA[919,39] := 1.0;
   DATA[920,0] := 2.538513;
   DATA[920,1] := 616.2683;
   DATA[920,2] := 2.0;
   DATA[920,3] := 1.0;
   DATA[920,4] := 262.5288;
   DATA[920,5] := 8.462446;
   DATA[920,6] := 315.4576;
   DATA[920,8] := 1.0;
   DATA[920,9] := 1.0;
   DATA[920,10] := 1.0;
   DATA[920,11] := 2.010372;
   DATA[920,13] := 1010.879;
   DATA[920,14] := 1.0;
   DATA[920,15] := 1.0;
   DATA[920,16] := 1.0;
   DATA[920,17] := 1.0;
   DATA[920,18] := 1.0;
   DATA[920,19] := 1.0;
   DATA[920,20] := 148.808;
   DATA[920,21] := 155.4217;
   DATA[920,22] := 1.71813;
   DATA[920,23] := 936.0292;
   DATA[920,24] := 2.0;
   DATA[920,25] := 2.0;
   DATA[920,26] := 7.878942;
   DATA[920,27] := 144.527;
   DATA[920,28] := 263.0415;
   DATA[920,29] := 12.07383;
   DATA[920,30] := 1.72443;
   DATA[920,31] := 1.274113;
   DATA[920,32] := 0.7353967;
   DATA[920,33] := 0.3084265;
   DATA[920,34] := 2.0;
   DATA[920,35] := 250.3204;
   DATA[920,36] := 1.681991;
   DATA[920,37] := 189.2464;
   DATA[920,38] := 0.000128152;
   DATA[920,39] := 1.0;
   DATA[921,0] := 2.542677;
   DATA[921,1] := 615.915;
   DATA[921,2] := 2.0;
   DATA[921,3] := 1.0;
   DATA[921,4] := 262.5288;
   DATA[921,5] := 8.462446;
   DATA[921,6] := 315.4576;
   DATA[921,8] := 1.0;
   DATA[921,9] := 1.0;
   DATA[921,10] := 1.0;
   DATA[921,11] := 2.010372;
   DATA[921,13] := 1010.718;
